LIN {X 0,Y 574.116,Z 389.505,A -85,B 0,C 180,E1 -2265.533,E2 -2265.533} C_VEL
LIN {X 0,Y 574.363,Z 374.82,A -85,B 0,C 180,E1 -2266.255,E2 -2266.255} C_VEL
LIN {X 0,Y 574.533,Z 360.604,A -85,B 0,C 180,E1 -2266.798,E2 -2266.798} C_VEL
LIN {X 0,Y 574.701,Z 345.577,A -85,B 0,C 180,E1 -2267.222,E2 -2267.222} C_VEL
LIN {X 0,Y 574.754,Z 330.659,A -85,B 0,C 180,E1 -2267.503,E2 -2267.503} C_VEL
LIN {X 0,Y 575.181,Z 176.218,A -85,B 0,C 180,E1 -2269.486,E2 -2269.486} C_VEL
LIN {X 0,Y 574.006,Z 169.785,A -85,B 0,C 180,E1 -2269.626,E2 -2269.626} C_VEL
LIN {X 0,Y 574.322,Z 144.284,A -85,B 0,C 180,E1 -2272.673,E2 -2272.673} C_VEL
LIN {X 0,Y 574.579,Z 122.188,A -85,B 0,C 180,E1 -2275.348,E2 -2275.348} C_VEL
LIN {X 0,Y 574.263,Z 119.027,A -85,B 0,C 180,E1 -2275.751,E2 -2275.751} C_VEL
LIN {X 0,Y 573.253,Z 114.708,A -85,B 0,C 180,E1 -2276.341,E2 -2276.341} C_VEL
LIN {X 0,Y 573.234,Z 114.705,A -85,B 0,C 180,E1 -2278.565,E2 -2278.565} C_VEL
LIN {X 0,Y 573.226,Z 114.702,A -85,B 0,C 180,E1 -2280.994,E2 -2280.994} C_VEL
LIN {X 0,Y 573.265,Z 114.701,A -85,B 0,C 180,E1 -2283.524,E2 -2283.524} C_VEL
LIN {X 0,Y 573.216,Z 114.711,A -85,B 0,C 180,E1 -2286.052,E2 -2286.052} C_VEL
LIN {X 0,Y 573.247,Z 114.699,A -85,B 0,C 180,E1 -2288.702,E2 -2288.702} C_VEL
LIN {X 0,Y 573.227,Z 114.709,A -85,B 0,C 180,E1 -2291.593,E2 -2291.593} C_VEL
LIN {X 0,Y 573.227,Z 114.703,A -85,B 0,C 180,E1 -2294.335,E2 -2294.335} C_VEL
LIN {X 0,Y 573.24,Z 114.707,A -85,B 0,C 180,E1 -2297.359,E2 -2297.359} C_VEL
LIN {X 0,Y 573.238,Z 114.699,A -85,B 0,C 180,E1 -2300.392,E2 -2300.392} C_VEL
LIN {X 0,Y 573.255,Z 114.703,A -85,B 0,C 180,E1 -2303.078,E2 -2303.078} C_VEL
LIN {X 0,Y 573.259,Z 114.701,A -85,B 0,C 180,E1 -2305.671,E2 -2305.671} C_VEL
LIN {X 0,Y 573.239,Z 114.699,A -85,B 0,C 180,E1 -2308.185,E2 -2308.185} C_VEL
LIN {X 0,Y 573.245,Z 114.701,A -85,B 0,C 180,E1 -2310.633,E2 -2310.633} C_VEL
LIN {X 0,Y 573.235,Z 114.701,A -85,B 0,C 180,E1 -2313.509,E2 -2313.509} C_VEL
LIN {X 0,Y 573.202,Z 114.704,A -85,B 0,C 180,E1 -2316.133,E2 -2316.133} C_VEL
LIN {X 0,Y 573.248,Z 114.703,A -85,B 0,C 180,E1 -2319.174,E2 -2319.174} C_VEL
LIN {X 0,Y 573.203,Z 114.705,A -85,B 0,C 180,E1 -2321.411,E2 -2321.411} C_VEL
LIN {X 0,Y 573.228,Z 114.7,A -85,B 0,C 180,E1 -2323.621,E2 -2323.621} C_VEL
LIN {X 0,Y 573.244,Z 114.699,A -85,B 0,C 180,E1 -2325.807,E2 -2325.807} C_VEL
LIN {X 0,Y 573.269,Z 114.702,A -85,B 0,C 180,E1 -2328.746,E2 -2328.746} C_VEL
LIN {X 0,Y 573.246,Z 114.698,A -85,B 0,C 180,E1 -2331.54,E2 -2331.54} C_VEL
LIN {X 0,Y 573.276,Z 114.705,A -85,B 0,C 180,E1 -2334.372,E2 -2334.372} C_VEL
LIN {X 0,Y 573.31,Z 114.693,A -85,B 0,C 180,E1 -2337.893,E2 -2337.893} C_VEL
LIN {X 0,Y 573.32,Z 114.692,A -85,B 0,C 180,E1 -2340,E2 -2340} C_VEL
LIN {X 0,Y 573.275,Z 114.695,A -85,B 0,C 180,E1 -2342.811,E2 -2342.811} C_VEL
LIN {X 0,Y 573.268,Z 114.699,A -85,B 0,C 180,E1 -2345.629,E2 -2345.629} C_VEL
LIN {X 0,Y 573.236,Z 114.698,A -85,B 0,C 180,E1 -2348.461,E2 -2348.461} C_VEL
LIN {X 0,Y 573.241,Z 114.699,A -85,B 0,C 180,E1 -2351.313,E2 -2351.313} C_VEL
LIN {X 0,Y 573.241,Z 114.7,A -85,B 0,C 180,E1 -2354.406,E2 -2354.406} C_VEL
LIN {X 0,Y 573.178,Z 114.708,A -85,B 0,C 180,E1 -2357.114,E2 -2357.114} C_VEL
LIN {X 0,Y 573.189,Z 114.708,A -85,B 0,C 180,E1 -2360.079,E2 -2360.079} C_VEL
LIN {X 0,Y 573.188,Z 114.705,A -85,B 0,C 180,E1 -2362.34,E2 -2362.34} C_VEL
LIN {X 0,Y 573.188,Z 114.706,A -85,B 0,C 180,E1 -2364.343,E2 -2364.343} C_VEL
LIN {X 0,Y 572.549,Z 114.789,A -85,B 0,C 180,E1 -2364.929,E2 -2364.929} C_VEL
LIN {X 0,Y 569.719,Z 115.148,A -85,B 0,C 180,E1 -2365.881,E2 -2365.881} C_VEL
LIN {X 0,Y 567.303,Z 115.452,A -85,B 0,C 180,E1 -2366.646,E2 -2366.646} C_VEL
LIN {X 0,Y 566.247,Z 115.579,A -85,B 0,C 180,E1 -2367.237,E2 -2367.237} C_VEL
LIN {X 0,Y 566.152,Z 115.587,A -85,B 0,C 180,E1 -2367.438,E2 -2367.438} C_VEL
LIN {X 0,Y 566.149,Z 115.582,A -85,B 0,C 180,E1 -2369.772,E2 -2369.772} C_VEL
LIN {X 0,Y 566.174,Z 115.579,A -85,B 0,C 180,E1 -2372.424,E2 -2372.424} C_VEL
LIN {X 0,Y 566.159,Z 115.589,A -85,B 0,C 180,E1 -2374.985,E2 -2374.985} C_VEL
LIN {X 0,Y 566.183,Z 115.578,A -85,B 0,C 180,E1 -2377.462,E2 -2377.462} C_VEL
LIN {X 0,Y 566.209,Z 115.574,A -85,B 0,C 180,E1 -2380.199,E2 -2380.199} C_VEL
LIN {X 0,Y 566.154,Z 115.588,A -85,B 0,C 180,E1 -2383.059,E2 -2383.059} C_VEL
LIN {X 0,Y 566.161,Z 115.579,A -85,B 0,C 180,E1 -2386.053,E2 -2386.053} C_VEL
LIN {X 0,Y 566.155,Z 115.589,A -85,B 0,C 180,E1 -2388.858,E2 -2388.858} C_VEL
LIN {X 0,Y 566.203,Z 115.575,A -85,B 0,C 180,E1 -2391.444,E2 -2391.444} C_VEL
LIN {X 0,Y 566.146,Z 115.589,A -85,B 0,C 180,E1 -2394.306,E2 -2394.306} C_VEL
LIN {X 0,Y 566.2,Z 115.577,A -85,B 0,C 180,E1 -2396.896,E2 -2396.896} C_VEL
LIN {X 0,Y 566.173,Z 115.58,A -85,B 0,C 180,E1 -2399.406,E2 -2399.406} C_VEL
LIN {X 0,Y 566.157,Z 115.585,A -85,B 0,C 180,E1 -2401.854,E2 -2401.854} C_VEL
LIN {X 0,Y 566.196,Z 115.586,A -85,B 0,C 180,E1 -2404.25,E2 -2404.25} C_VEL
LIN {X 0,Y 566.168,Z 115.582,A -85,B 0,C 180,E1 -2407.368,E2 -2407.368} C_VEL
LIN {X 0,Y 566.206,Z 115.58,A -85,B 0,C 180,E1 -2409.662,E2 -2409.662} C_VEL
LIN {X 0,Y 566.18,Z 115.585,A -85,B 0,C 180,E1 -2411.921,E2 -2411.921} C_VEL
LIN {X 0,Y 566.193,Z 115.578,A -85,B 0,C 180,E1 -2414.89,E2 -2414.89} C_VEL
LIN {X 0,Y 566.236,Z 115.581,A -85,B 0,C 180,E1 -2417.819,E2 -2417.819} C_VEL
LIN {X 0,Y 566.176,Z 115.586,A -85,B 0,C 180,E1 -2419.992,E2 -2419.992} C_VEL
LIN {X 0,Y 566.216,Z 115.577,A -85,B 0,C 180,E1 -2422.87,E2 -2422.87} C_VEL
LIN {X 0,Y 566.211,Z 115.616,A -85,B 0,C 180,E1 -2425.528,E2 -2425.528} C_VEL
LIN {X 0,Y 567.254,Z 121.648,A -85,B 0,C 180,E1 -2426.448,E2 -2426.448} C_VEL
LIN {X 0,Y 566.93,Z 140.906,A -85,B 0,C 180,E1 -2429.178,E2 -2429.178} C_VEL
LIN {X 0,Y 568.458,Z 149.206,A -85,B 0,C 180,E1 -2429.358,E2 -2429.358} C_VEL
LIN {X 0,Y 567.998,Z 306.402,A -85,B 0,C 180,E1 -2431.418,E2 -2431.418} C_VEL
LIN {X 0,Y 567.821,Z 322.005,A -85,B 0,C 180,E1 -2431.773,E2 -2431.773} C_VEL
LIN {X 0,Y 567.594,Z 336.9,A -85,B 0,C 180,E1 -2432.262,E2 -2432.262} C_VEL
LIN {X 0,Y 567.373,Z 352.096,A -85,B 0,C 180,E1 -2432.929,E2 -2432.929} C_VEL
LIN {X 0,Y 567.124,Z 365.069,A -85,B 0,C 180,E1 -2433.641,E2 -2433.641} C_VEL
LIN {X 0,Y 566.895,Z 378.339,A -85,B 0,C 180,E1 -2434.533,E2 -2434.533} C_VEL
LIN {X 0,Y 566.64,Z 390.468,A -85,B 0,C 180,E1 -2435.516,E2 -2435.516} C_VEL
LIN {X 0,Y 566.457,Z 401.276,A -85,B 0,C 180,E1 -2436.559,E2 -2436.559} C_VEL
LIN {X 0,Y 566.314,Z 410.997,A -85,B 0,C 180,E1 -2437.666,E2 -2437.666} C_VEL
LIN {X 0,Y 566.184,Z 420.325,A -85,B 0,C 180,E1 -2438.926,E2 -2438.926} C_VEL
LIN {X 0,Y 566.046,Z 428.145,A -85,B 0,C 180,E1 -2440.191,E2 -2440.191} C_VEL
LIN {X 0,Y 565.957,Z 434.669,A -85,B 0,C 180,E1 -2441.46,E2 -2441.46} C_VEL
LIN {X 0,Y 565.907,Z 440.687,A -85,B 0,C 180,E1 -2442.917,E2 -2442.917} C_VEL
LIN {X 0,Y 565.884,Z 445.316,A -85,B 0,C 180,E1 -2444.382,E2 -2444.382} C_VEL
LIN {X 0,Y 565.827,Z 448.637,A -85,B 0,C 180,E1 -2445.858,E2 -2445.858} C_VEL
LIN {X 0,Y 565.833,Z 450.67,A -85,B 0,C 180,E1 -2447.343,E2 -2447.343} C_VEL
LIN {X 0,Y 565.852,Z 451.461,A -85,B 0,C 180,E1 -2448.84,E2 -2448.84} C_VEL
LIN {X 0,Y 565.823,Z 450.989,A -85,B 0,C 180,E1 -2450.352,E2 -2450.352} C_VEL
LIN {X 0,Y 565.835,Z 449.211,A -85,B 0,C 180,E1 -2451.877,E2 -2451.877} C_VEL
LIN {X 0,Y 565.894,Z 446.046,A -85,B 0,C 180,E1 -2453.417,E2 -2453.417} C_VEL
LIN {X 0,Y 565.927,Z 441.37,A -85,B 0,C 180,E1 -2454.975,E2 -2454.975} C_VEL
LIN {X 0,Y 565.969,Z 436.799,A -85,B 0,C 180,E1 -2456.156,E2 -2456.156} C_VEL
LIN {X 0,Y 566.03,Z 430.112,A -85,B 0,C 180,E1 -2457.549,E2 -2457.549} C_VEL
LIN {X 0,Y 566.16,Z 421.756,A -85,B 0,C 180,E1 -2458.955,E2 -2458.955} C_VEL
LIN {X 0,Y 566.299,Z 413.022,A -85,B 0,C 180,E1 -2460.173,E2 -2460.173} C_VEL
LIN {X 0,Y 566.444,Z 402.483,A -85,B 0,C 180,E1 -2461.406,E2 -2461.406} C_VEL
LIN {X 0,Y 566.662,Z 390.517,A -85,B 0,C 180,E1 -2462.569,E2 -2462.569} C_VEL
LIN {X 0,Y 566.897,Z 377.894,A -85,B 0,C 180,E1 -2463.589,E2 -2463.589} C_VEL
LIN {X 0,Y 567.109,Z 365.372,A -85,B 0,C 180,E1 -2464.431,E2 -2464.431} C_VEL
LIN {X 0,Y 567.374,Z 352.119,A -85,B 0,C 180,E1 -2465.161,E2 -2465.161} C_VEL
LIN {X 0,Y 567.602,Z 337.434,A -85,B 0,C 180,E1 -2465.806,E2 -2465.806} C_VEL
LIN {X 0,Y 567.825,Z 322.2,A -85,B 0,C 180,E1 -2466.311,E2 -2466.311} C_VEL
LIN {X 0,Y 567.967,Z 306.458,A -85,B 0,C 180,E1 -2466.672,E2 -2466.672} C_VEL
LIN {X 0,Y 568.468,Z 148.223,A -85,B 0,C 180,E1 -2468.745,E2 -2468.745} C_VEL
LIN {X 0,Y 566.907,Z 140.941,A -85,B 0,C 180,E1 -2468.909,E2 -2468.909} C_VEL
LIN {X 0,Y 567.252,Z 121.495,A -85,B 0,C 180,E1 -2471.67,E2 -2471.67} C_VEL
LIN {X 0,Y 566.185,Z 115.588,A -85,B 0,C 180,E1 -2472.599,E2 -2472.599} C_VEL
LIN {X 0,Y 566.166,Z 115.585,A -85,B 0,C 180,E1 -2475.036,E2 -2475.036} C_VEL
LIN {X 0,Y 566.178,Z 115.584,A -85,B 0,C 180,E1 -2477.909,E2 -2477.909} C_VEL
LIN {X 0,Y 566.212,Z 115.582,A -85,B 0,C 180,E1 -2480.726,E2 -2480.726} C_VEL
LIN {X 0,Y 566.184,Z 115.58,A -85,B 0,C 180,E1 -2483.428,E2 -2483.428} C_VEL
LIN {X 0,Y 566.213,Z 115.585,A -85,B 0,C 180,E1 -2486.266,E2 -2486.266} C_VEL
LIN {X 0,Y 566.186,Z 115.579,A -85,B 0,C 180,E1 -2488.924,E2 -2488.924} C_VEL
LIN {X 0,Y 566.192,Z 115.583,A -85,B 0,C 180,E1 -2491.856,E2 -2491.856} C_VEL
LIN {X 0,Y 566.197,Z 115.582,A -85,B 0,C 180,E1 -2494.25,E2 -2494.25} C_VEL
LIN {X 0,Y 566.167,Z 115.58,A -85,B 0,C 180,E1 -2496.72,E2 -2496.72} C_VEL
LIN {X 0,Y 566.206,Z 115.582,A -85,B 0,C 180,E1 -2499.662,E2 -2499.662} C_VEL
LIN {X 0,Y 566.18,Z 115.587,A -85,B 0,C 180,E1 -2501.921,E2 -2501.921} C_VEL
LIN {X 0,Y 566.191,Z 115.577,A -85,B 0,C 180,E1 -2504.89,E2 -2504.89} C_VEL
LIN {X 0,Y 566.234,Z 115.58,A -85,B 0,C 180,E1 -2507.819,E2 -2507.819} C_VEL
LIN {X 0,Y 566.178,Z 115.583,A -85,B 0,C 180,E1 -2509.992,E2 -2509.992} C_VEL
LIN {X 0,Y 566.242,Z 115.572,A -85,B 0,C 180,E1 -2512.87,E2 -2512.87} C_VEL
LIN {X 0,Y 566.277,Z 115.568,A -85,B 0,C 180,E1 -2515.016,E2 -2515.016} C_VEL
LIN {X 0,Y 566.287,Z 115.568,A -85,B 0,C 180,E1 -2517.866,E2 -2517.866} C_VEL
LIN {X 0,Y 566.293,Z 115.566,A -85,B 0,C 180,E1 -2520.711,E2 -2520.711} C_VEL
LIN {X 0,Y 566.263,Z 115.571,A -85,B 0,C 180,E1 -2522.845,E2 -2522.845} C_VEL
LIN {X 0,Y 566.265,Z 115.571,A -85,B 0,C 180,E1 -2525.698,E2 -2525.698} C_VEL
LIN {X 0,Y 566.205,Z 115.577,A -85,B 0,C 180,E1 -2528.566,E2 -2528.566} C_VEL
LIN {X 0,Y 566.243,Z 115.575,A -85,B 0,C 180,E1 -2531.454,E2 -2531.454} C_VEL
LIN {X 0,Y 566.235,Z 115.575,A -85,B 0,C 180,E1 -2534.506,E2 -2534.506} C_VEL
LIN {X 0,Y 566.196,Z 115.581,A -85,B 0,C 180,E1 -2537.331,E2 -2537.331} C_VEL
LIN {X 0,Y 566.206,Z 115.577,A -85,B 0,C 180,E1 -2540.337,E2 -2540.337} C_VEL
LIN {X 0,Y 566.171,Z 115.583,A -85,B 0,C 180,E1 -2543.281,E2 -2543.281} C_VEL
LIN {X 0,Y 566.209,Z 115.575,A -85,B 0,C 180,E1 -2545.749,E2 -2545.749} C_VEL
LIN {X 0,Y 566.202,Z 115.579,A -85,B 0,C 180,E1 -2548.202,E2 -2548.202} C_VEL
LIN {X 0,Y 566.189,Z 115.58,A -85,B 0,C 180,E1 -2551.076,E2 -2551.076} C_VEL
LIN {X 0,Y 566.196,Z 115.578,A -85,B 0,C 180,E1 -2553.732,E2 -2553.732} C_VEL
LIN {X 0,Y 566.199,Z 115.584,A -85,B 0,C 180,E1 -2556.57,E2 -2556.57} C_VEL
LIN {X 0,Y 566.214,Z 115.574,A -85,B 0,C 180,E1 -2559.686,E2 -2559.686} C_VEL
LIN {X 0,Y 566.202,Z 115.576,A -85,B 0,C 180,E1 -2562.917,E2 -2562.917} C_VEL
LIN {X 0,Y 566.198,Z 115.584,A -85,B 0,C 180,E1 -2566.049,E2 -2566.049} C_VEL
LIN {X 0,Y 566.203,Z 115.576,A -85,B 0,C 180,E1 -2569.215,E2 -2569.215} C_VEL
LIN {X 0,Y 566.188,Z 115.582,A -85,B 0,C 180,E1 -2571.637,E2 -2571.637} C_VEL
LIN {X 0,Y 566.161,Z 115.586,A -85,B 0,C 180,E1 -2574.308,E2 -2574.308} C_VEL
LIN {X 0,Y 566.219,Z 115.574,A -85,B 0,C 180,E1 -2576.898,E2 -2576.898} C_VEL
LIN {X 0,Y 566.18,Z 115.583,A -85,B 0,C 180,E1 -2579.407,E2 -2579.407} C_VEL
LIN {X 0,Y 566.211,Z 115.584,A -85,B 0,C 180,E1 -2581.858,E2 -2581.858} C_VEL
LIN {X 0,Y 566.206,Z 115.624,A -85,B 0,C 180,E1 -2583.459,E2 -2583.459} C_VEL
LIN {X 0,Y 567.659,Z 121.967,A -85,B 0,C 180,E1 -2584.322,E2 -2584.322} C_VEL
LIN {X 0,Y 567.503,Z 140.923,A -85,B 0,C 180,E1 -2586.654,E2 -2586.654} C_VEL
LIN {X 0,Y 567.154,Z 164.6,A -85,B 0,C 180,E1 -2589.509,E2 -2589.509} C_VEL
LIN {X 0,Y 567.115,Z 169.895,A -85,B 0,C 180,E1 -2590.142,E2 -2590.142} C_VEL
LIN {X 0,Y 568.508,Z 178.337,A -85,B 0,C 180,E1 -2590.304,E2 -2590.304} C_VEL
LIN {X 0,Y 567.984,Z 335.946,A -85,B 0,C 180,E1 -2592.364,E2 -2592.364} C_VEL
LIN {X 0,Y 567.834,Z 351.709,A -85,B 0,C 180,E1 -2592.72,E2 -2592.72} C_VEL
LIN {X 0,Y 567.616,Z 367.04,A -85,B 0,C 180,E1 -2593.223,E2 -2593.223} C_VEL
LIN {X 0,Y 567.453,Z 380.783,A -85,B 0,C 180,E1 -2593.82,E2 -2593.82} C_VEL
LIN {X 0,Y 567.154,Z 394.255,A -85,B 0,C 180,E1 -2594.549,E2 -2594.549} C_VEL
LIN {X 0,Y 566.931,Z 406.522,A -85,B 0,C 180,E1 -2595.359,E2 -2595.359} C_VEL
LIN {X 0,Y 566.672,Z 419.296,A -85,B 0,C 180,E1 -2596.371,E2 -2596.371} C_VEL
LIN {X 0,Y 566.491,Z 430.752,A -85,B 0,C 180,E1 -2597.461,E2 -2597.461} C_VEL
LIN {X 0,Y 566.268,Z 441.313,A -85,B 0,C 180,E1 -2598.659,E2 -2598.659} C_VEL
LIN {X 0,Y 566.208,Z 449.857,A -85,B 0,C 180,E1 -2599.812,E2 -2599.812} C_VEL
LIN {X 0,Y 566.057,Z 457.737,A -85,B 0,C 180,E1 -2601.072,E2 -2601.072} C_VEL
LIN {X 0,Y 565.997,Z 465.091,A -85,B 0,C 180,E1 -2602.509,E2 -2602.509} C_VEL
LIN {X 0,Y 565.959,Z 470.923,A -85,B 0,C 180,E1 -2603.941,E2 -2603.941} C_VEL
LIN {X 0,Y 565.866,Z 474.387,A -85,B 0,C 180,E1 -2605.013,E2 -2605.013} C_VEL
LIN {X 0,Y 565.91,Z 477.89,A -85,B 0,C 180,E1 -2606.44,E2 -2606.44} C_VEL
LIN {X 0,Y 565.839,Z 480.191,A -85,B 0,C 180,E1 -2607.865,E2 -2607.865} C_VEL
LIN {X 0,Y 565.837,Z 481.349,A -85,B 0,C 180,E1 -2609.289,E2 -2609.289} C_VEL
LIN {X 0,Y 565.837,Z 481.348,A -85,B 0,C 180,E1 -2610.712,E2 -2610.712} C_VEL
LIN {X 0,Y 565.839,Z 480.188,A -85,B 0,C 180,E1 -2612.136,E2 -2612.136} C_VEL
LIN {X 0,Y 565.91,Z 477.885,A -85,B 0,C 180,E1 -2613.56,E2 -2613.56} C_VEL
LIN {X 0,Y 565.867,Z 474.385,A -85,B 0,C 180,E1 -2614.988,E2 -2614.988} C_VEL
LIN {X 0,Y 565.943,Z 469.607,A -85,B 0,C 180,E1 -2616.417,E2 -2616.417} C_VEL
LIN {X 0,Y 566.014,Z 463.42,A -85,B 0,C 180,E1 -2617.85,E2 -2617.85} C_VEL
LIN {X 0,Y 566.071,Z 455.644,A -85,B 0,C 180,E1 -2619.289,E2 -2619.289} C_VEL
LIN {X 0,Y 566.239,Z 447.365,A -85,B 0,C 180,E1 -2620.549,E2 -2620.549} C_VEL
LIN {X 0,Y 566.368,Z 437.388,A -85,B 0,C 180,E1 -2621.815,E2 -2621.815} C_VEL
LIN {X 0,Y 566.586,Z 427.183,A -85,B 0,C 180,E1 -2622.902,E2 -2622.902} C_VEL
LIN {X 0,Y 566.8,Z 415.015,A -85,B 0,C 180,E1 -2623.992,E2 -2623.992} C_VEL
LIN {X 0,Y 567.038,Z 402.332,A -85,B 0,C 180,E1 -2624.937,E2 -2624.937} C_VEL
LIN {X 0,Y 567.235,Z 389.501,A -85,B 0,C 180,E1 -2625.726,E2 -2625.726} C_VEL
LIN {X 0,Y 567.497,Z 374.816,A -85,B 0,C 180,E1 -2626.457,E2 -2626.457} C_VEL
LIN {X 0,Y 567.721,Z 360.603,A -85,B 0,C 180,E1 -2627.006,E2 -2627.006} C_VEL
LIN {X 0,Y 567.923,Z 346.228,A -85,B 0,C 180,E1 -2627.418,E2 -2627.418} C_VEL
LIN {X 0,Y 567.984,Z 331.773,A -85,B 0,C 180,E1 -2627.701,E2 -2627.701} C_VEL
LIN {X 0,Y 568.459,Z 176.883,A -85,B 0,C 180,E1 -2629.717,E2 -2629.717} C_VEL
LIN {X 0,Y 567.12,Z 169.805,A -85,B 0,C 180,E1 -2629.868,E2 -2629.868} C_VEL
LIN {X 0,Y 567.438,Z 145.69,A -85,B 0,C 180,E1 -2632.771,E2 -2632.771} C_VEL
LIN {X 0,Y 567.746,Z 123.819,A -85,B 0,C 180,E1 -2635.451,E2 -2635.451} C_VEL
LIN {X 0,Y 567,Z 118.863,A -85,B 0,C 180,E1 -2636.106,E2 -2636.106} C_VEL
LIN {X 0,Y 566.215,Z 115.583,A -85,B 0,C 180,E1 -2636.584,E2 -2636.584} C_VEL
LIN {X 0,Y 566.189,Z 115.58,A -85,B 0,C 180,E1 -2638.954,E2 -2638.954} C_VEL
LIN {X 0,Y 566.194,Z 115.58,A -85,B 0,C 180,E1 -2641.422,E2 -2641.422} C_VEL
LIN {X 0,Y 566.211,Z 115.585,A -85,B 0,C 180,E1 -2643.956,E2 -2643.956} C_VEL
LIN {X 0,Y 566.201,Z 115.579,A -85,B 0,C 180,E1 -2646.57,E2 -2646.57} C_VEL
LIN {X 0,Y 566.223,Z 115.582,A -85,B 0,C 180,E1 -2649.687,E2 -2649.687} C_VEL
LIN {X 0,Y 566.2,Z 115.577,A -85,B 0,C 180,E1 -2652.917,E2 -2652.917} C_VEL
LIN {X 0,Y 566.197,Z 115.581,A -85,B 0,C 180,E1 -2656.05,E2 -2656.05} C_VEL
LIN {X 0,Y 566.206,Z 115.582,A -85,B 0,C 180,E1 -2659.215,E2 -2659.215} C_VEL
LIN {X 0,Y 566.183,Z 115.584,A -85,B 0,C 180,E1 -2661.637,E2 -2661.637} C_VEL
LIN {X 0,Y 566.164,Z 115.581,A -85,B 0,C 180,E1 -2664.308,E2 -2664.308} C_VEL
LIN {X 0,Y 566.202,Z 115.581,A -85,B 0,C 180,E1 -2666.897,E2 -2666.897} C_VEL
LIN {X 0,Y 566.172,Z 115.585,A -85,B 0,C 180,E1 -2669.407,E2 -2669.407} C_VEL
LIN {X 0,Y 566.173,Z 115.577,A -85,B 0,C 180,E1 -2671.856,E2 -2671.856} C_VEL
LIN {X 0,Y 566.204,Z 115.575,A -85,B 0,C 180,E1 -2674.251,E2 -2674.251} C_VEL
LIN {X 0,Y 566.166,Z 115.583,A -85,B 0,C 180,E1 -2677.368,E2 -2677.368} C_VEL
LIN {X 0,Y 566.204,Z 115.576,A -85,B 0,C 180,E1 -2679.663,E2 -2679.663} C_VEL
LIN {X 0,Y 566.177,Z 115.579,A -85,B 0,C 180,E1 -2681.921,E2 -2681.921} C_VEL
LIN {X 0,Y 566.184,Z 115.58,A -85,B 0,C 180,E1 -2684.152,E2 -2684.152} C_VEL
LIN {X 0,Y 566.171,Z 115.585,A -85,B 0,C 180,E1 -2686.358,E2 -2686.358} C_VEL
LIN {X 0,Y 566.236,Z 115.573,A -85,B 0,C 180,E1 -2689.271,E2 -2689.271} C_VEL
LIN {X 0,Y 566.209,Z 115.58,A -85,B 0,C 180,E1 -2692.153,E2 -2692.153} C_VEL
LIN {X 0,Y 566.256,Z 115.57,A -85,B 0,C 180,E1 -2695.016,E2 -2695.016} C_VEL
LIN {X 0,Y 566.28,Z 115.568,A -85,B 0,C 180,E1 -2697.867,E2 -2697.867} C_VEL
LIN {X 0,Y 566.289,Z 115.567,A -85,B 0,C 180,E1 -2700,E2 -2700} C_VEL
LIN {X 0,Y 566.243,Z 115.571,A -85,B 0,C 180,E1 -2702.846,E2 -2702.846} C_VEL
LIN {X 0,Y 566.237,Z 115.576,A -85,B 0,C 180,E1 -2705.699,E2 -2705.699} C_VEL
LIN {X 0,Y 566.188,Z 115.575,A -85,B 0,C 180,E1 -2708.567,E2 -2708.567} C_VEL
LIN {X 0,Y 566.197,Z 115.577,A -85,B 0,C 180,E1 -2711.456,E2 -2711.456} C_VEL
LIN {X 0,Y 566.188,Z 115.578,A -85,B 0,C 180,E1 -2714.486,E2 -2714.486} C_VEL
LIN {X 0,Y 566.152,Z 115.586,A -85,B 0,C 180,E1 -2717.334,E2 -2717.334} C_VEL
LIN {X 0,Y 566.14,Z 115.584,A -85,B 0,C 180,E1 -2720.34,E2 -2720.34} C_VEL
LIN {X 0,Y 566.135,Z 115.584,A -85,B 0,C 180,E1 -2722.634,E2 -2722.634} C_VEL
LIN {X 0,Y 566.147,Z 115.587,A -85,B 0,C 180,E1 -2725.013,E2 -2725.013} C_VEL
LIN {X 0,Y 566.152,Z 115.587,A -85,B 0,C 180,E1 -2727.438,E2 -2727.438} C_VEL
LIN {X 0,Y 565.458,Z 115.669,A -85,B 0,C 180,E1 -2728.032,E2 -2728.032} C_VEL
LIN {X 0,Y 562.584,Z 116.028,A -85,B 0,C 180,E1 -2728.995,E2 -2728.995} C_VEL
LIN {X 0,Y 560.184,Z 116.324,A -85,B 0,C 180,E1 -2729.771,E2 -2729.771} C_VEL
LIN {X 0,Y 559.173,Z 116.448,A -85,B 0,C 180,E1 -2730.37,E2 -2730.37} C_VEL
LIN {X 0,Y 559.101,Z 116.458,A -85,B 0,C 180,E1 -2730.573,E2 -2730.573} C_VEL
LIN {X 0,Y 559.137,Z 116.458,A -85,B 0,C 180,E1 -2732.717,E2 -2732.717} C_VEL
LIN {X 0,Y 559.114,Z 116.464,A -85,B 0,C 180,E1 -2735.326,E2 -2735.326} C_VEL
LIN {X 0,Y 559.111,Z 116.455,A -85,B 0,C 180,E1 -2738.02,E2 -2738.02} C_VEL
LIN {X 0,Y 559.159,Z 116.452,A -85,B 0,C 180,E1 -2739.941,E2 -2739.941} C_VEL
LIN {X 0,Y 559.105,Z 116.464,A -85,B 0,C 180,E1 -2743.191,E2 -2743.191} C_VEL
LIN {X 0,Y 559.128,Z 116.453,A -85,B 0,C 180,E1 -2745.764,E2 -2745.764} C_VEL
LIN {X 0,Y 559.105,Z 116.462,A -85,B 0,C 180,E1 -2748.224,E2 -2748.224} C_VEL
LIN {X 0,Y 559.172,Z 116.452,A -85,B 0,C 180,E1 -2751.193,E2 -2751.193} C_VEL
LIN {X 0,Y 559.122,Z 116.458,A -85,B 0,C 180,E1 -2753.787,E2 -2753.787} C_VEL
LIN {X 0,Y 559.15,Z 116.463,A -85,B 0,C 180,E1 -2756.424,E2 -2756.424} C_VEL
LIN {X 0,Y 559.154,Z 116.456,A -85,B 0,C 180,E1 -2758.98,E2 -2758.98} C_VEL
LIN {X 0,Y 559.117,Z 116.46,A -85,B 0,C 180,E1 -2761.63,E2 -2761.63} C_VEL
LIN {X 0,Y 559.162,Z 116.459,A -85,B 0,C 180,E1 -2763.902,E2 -2763.902} C_VEL
LIN {X 0,Y 559.117,Z 116.459,A -85,B 0,C 180,E1 -2767.066,E2 -2767.066} C_VEL
LIN {X 0,Y 559.177,Z 116.453,A -85,B 0,C 180,E1 -2769.395,E2 -2769.395} C_VEL
LIN {X 0,Y 559.129,Z 116.462,A -85,B 0,C 180,E1 -2771.685,E2 -2771.685} C_VEL
LIN {X 0,Y 559.144,Z 116.465,A -85,B 0,C 180,E1 -2773.947,E2 -2773.947} C_VEL
LIN {X 0,Y 559.165,Z 116.457,A -85,B 0,C 180,E1 -2776.184,E2 -2776.184} C_VEL
LIN {X 0,Y 559.197,Z 116.452,A -85,B 0,C 180,E1 -2779.133,E2 -2779.133} C_VEL
LIN {X 0,Y 559.195,Z 116.455,A -85,B 0,C 180,E1 -2782.053,E2 -2782.053} C_VEL
LIN {X 0,Y 559.252,Z 116.449,A -85,B 0,C 180,E1 -2784.953,E2 -2784.953} C_VEL
LIN {X 0,Y 559.215,Z 116.594,A -85,B 0,C 180,E1 -2785.337,E2 -2785.337} C_VEL
LIN {X 0,Y 560.328,Z 122.289,A -85,B 0,C 180,E1 -2786.224,E2 -2786.224} C_VEL
LIN {X 0,Y 560.049,Z 141.154,A -85,B 0,C 180,E1 -2788.936,E2 -2788.936} C_VEL
LIN {X 0,Y 561.748,Z 149.207,A -85,B 0,C 180,E1 -2789.111,E2 -2789.111} C_VEL
LIN {X 0,Y 561.251,Z 305.85,A -85,B 0,C 180,E1 -2791.188,E2 -2791.188} C_VEL
LIN {X 0,Y 561.068,Z 321.67,A -85,B 0,C 180,E1 -2791.547,E2 -2791.547} C_VEL
LIN {X 0,Y 560.799,Z 337.211,A -85,B 0,C 180,E1 -2792.065,E2 -2792.065} C_VEL
LIN {X 0,Y 560.541,Z 351.484,A -85,B 0,C 180,E1 -2792.695,E2 -2792.695} C_VEL
LIN {X 0,Y 560.244,Z 364.549,A -85,B 0,C 180,E1 -2793.416,E2 -2793.416} C_VEL
LIN {X 0,Y 560.029,Z 377.892,A -85,B 0,C 180,E1 -2794.318,E2 -2794.318} C_VEL
LIN {X 0,Y 559.712,Z 390.106,A -85,B 0,C 180,E1 -2795.313,E2 -2795.313} C_VEL
LIN {X 0,Y 559.438,Z 402.159,A -85,B 0,C 180,E1 -2796.492,E2 -2796.492} C_VEL
LIN {X 0,Y 559.267,Z 412.938,A -85,B 0,C 180,E1 -2797.764,E2 -2797.764} C_VEL
LIN {X 0,Y 559.104,Z 421.959,A -85,B 0,C 180,E1 -2799.04,E2 -2799.04} C_VEL
LIN {X 0,Y 558.953,Z 429.492,A -85,B 0,C 180,E1 -2800.321,E2 -2800.321} C_VEL
LIN {X 0,Y 558.868,Z 435.753,A -85,B 0,C 180,E1 -2801.607,E2 -2801.607} C_VEL
LIN {X 0,Y 558.819,Z 441.525,A -85,B 0,C 180,E1 -2803.084,E2 -2803.084} C_VEL
LIN {X 0,Y 558.787,Z 445.923,A -85,B 0,C 180,E1 -2804.569,E2 -2804.569} C_VEL
LIN {X 0,Y 558.741,Z 449.031,A -85,B 0,C 180,E1 -2806.064,E2 -2806.064} C_VEL
LIN {X 0,Y 558.748,Z 450.886,A -85,B 0,C 180,E1 -2807.57,E2 -2807.57} C_VEL
LIN {X 0,Y 558.78,Z 451.497,A -85,B 0,C 180,E1 -2809.087,E2 -2809.087} C_VEL
LIN {X 0,Y 558.738,Z 450.819,A -85,B 0,C 180,E1 -2810.621,E2 -2810.621} C_VEL
LIN {X 0,Y 558.749,Z 448.812,A -85,B 0,C 180,E1 -2812.169,E2 -2812.169} C_VEL
LIN {X 0,Y 558.821,Z 445.404,A -85,B 0,C 180,E1 -2813.731,E2 -2813.731} C_VEL
LIN {X 0,Y 558.857,Z 440.469,A -85,B 0,C 180,E1 -2815.313,E2 -2815.313} C_VEL
LIN {X 0,Y 558.918,Z 434.455,A -85,B 0,C 180,E1 -2816.775,E2 -2816.775} C_VEL
LIN {X 0,Y 559.003,Z 427.997,A -85,B 0,C 180,E1 -2818.039,E2 -2818.039} C_VEL
LIN {X 0,Y 559.124,Z 419.913,A -85,B 0,C 180,E1 -2819.355,E2 -2819.355} C_VEL
LIN {X 0,Y 559.297,Z 410.81,A -85,B 0,C 180,E1 -2820.591,E2 -2820.591} C_VEL
LIN {X 0,Y 559.499,Z 399.803,A -85,B 0,C 180,E1 -2821.841,E2 -2821.841} C_VEL
LIN {X 0,Y 559.749,Z 388.032,A -85,B 0,C 180,E1 -2822.955,E2 -2822.955} C_VEL
LIN {X 0,Y 560.033,Z 376.418,A -85,B 0,C 180,E1 -2823.878,E2 -2823.878} C_VEL
LIN {X 0,Y 560.268,Z 364.22,A -85,B 0,C 180,E1 -2824.693,E2 -2824.693} C_VEL
LIN {X 0,Y 560.579,Z 350.088,A -85,B 0,C 180,E1 -2825.462,E2 -2825.462} C_VEL
LIN {X 0,Y 560.793,Z 335.596,A -85,B 0,C 180,E1 -2826.087,E2 -2826.087} C_VEL
LIN {X 0,Y 561.047,Z 320.66,A -85,B 0,C 180,E1 -2826.57,E2 -2826.57} C_VEL
LIN {X 0,Y 561.214,Z 306.017,A -85,B 0,C 180,E1 -2826.9,E2 -2826.9} C_VEL
LIN {X 0,Y 561.786,Z 149.464,A -85,B 0,C 180,E1 -2828.974,E2 -2828.974} C_VEL
LIN {X 0,Y 560.008,Z 141.228,A -85,B 0,C 180,E1 -2829.152,E2 -2829.152} C_VEL
LIN {X 0,Y 560.394,Z 123.75,A -85,B 0,C 180,E1 -2831.658,E2 -2831.658} C_VEL
LIN {X 0,Y 559.526,Z 118.2,A -85,B 0,C 180,E1 -2832.512,E2 -2832.512} C_VEL
LIN {X 0,Y 559.155,Z 116.463,A -85,B 0,C 180,E1 -2832.792,E2 -2832.792} C_VEL
LIN {X 0,Y 559.149,Z 116.458,A -85,B 0,C 180,E1 -2835.761,E2 -2835.761} C_VEL
LIN {X 0,Y 559.157,Z 116.462,A -85,B 0,C 180,E1 -2838.229,E2 -2838.229} C_VEL
LIN {X 0,Y 559.173,Z 116.455,A -85,B 0,C 180,E1 -2841.192,E2 -2841.192} C_VEL
LIN {X 0,Y 559.123,Z 116.462,A -85,B 0,C 180,E1 -2843.787,E2 -2843.787} C_VEL
LIN {X 0,Y 559.164,Z 116.46,A -85,B 0,C 180,E1 -2846.425,E2 -2846.425} C_VEL
LIN {X 0,Y 559.151,Z 116.455,A -85,B 0,C 180,E1 -2848.98,E2 -2848.98} C_VEL
LIN {X 0,Y 559.146,Z 116.457,A -85,B 0,C 180,E1 -2851.623,E2 -2851.623} C_VEL
LIN {X 0,Y 559.163,Z 116.461,A -85,B 0,C 180,E1 -2853.902,E2 -2853.902} C_VEL
LIN {X 0,Y 559.12,Z 116.457,A -85,B 0,C 180,E1 -2857.066,E2 -2857.066} C_VEL
LIN {X 0,Y 559.176,Z 116.454,A -85,B 0,C 180,E1 -2859.395,E2 -2859.395} C_VEL
LIN {X 0,Y 559.129,Z 116.465,A -85,B 0,C 180,E1 -2861.685,E2 -2861.685} C_VEL
LIN {X 0,Y 559.147,Z 116.462,A -85,B 0,C 180,E1 -2863.947,E2 -2863.947} C_VEL
LIN {X 0,Y 559.162,Z 116.457,A -85,B 0,C 180,E1 -2866.183,E2 -2866.183} C_VEL
LIN {X 0,Y 559.196,Z 116.451,A -85,B 0,C 180,E1 -2869.133,E2 -2869.133} C_VEL
LIN {X 0,Y 559.199,Z 116.452,A -85,B 0,C 180,E1 -2872.053,E2 -2872.053} C_VEL
LIN {X 0,Y 559.251,Z 116.443,A -85,B 0,C 180,E1 -2874.953,E2 -2874.953} C_VEL
LIN {X 0,Y 559.258,Z 116.444,A -85,B 0,C 180,E1 -2877.839,E2 -2877.839} C_VEL
LIN {X 0,Y 559.265,Z 116.442,A -85,B 0,C 180,E1 -2880.72,E2 -2880.72} C_VEL
LIN {X 0,Y 559.231,Z 116.447,A -85,B 0,C 180,E1 -2882.881,E2 -2882.881} C_VEL
LIN {X 0,Y 559.233,Z 116.446,A -85,B 0,C 180,E1 -2885.77,E2 -2885.77} C_VEL
LIN {X 0,Y 559.17,Z 116.454,A -85,B 0,C 180,E1 -2888.674,E2 -2888.674} C_VEL
LIN {X 0,Y 559.206,Z 116.449,A -85,B 0,C 180,E1 -2891.6,E2 -2891.6} C_VEL
LIN {X 0,Y 559.201,Z 116.452,A -85,B 0,C 180,E1 -2894.595,E2 -2894.595} C_VEL
LIN {X 0,Y 559.14,Z 116.458,A -85,B 0,C 180,E1 -2897.557,E2 -2897.557} C_VEL
LIN {X 0,Y 559.165,Z 116.452,A -85,B 0,C 180,E1 -2899.837,E2 -2899.837} C_VEL
LIN {X 0,Y 559.14,Z 116.457,A -85,B 0,C 180,E1 -2902.153,E2 -2902.153} C_VEL
LIN {X 0,Y 559.175,Z 116.453,A -85,B 0,C 180,E1 -2905.298,E2 -2905.298} C_VEL
LIN {X 0,Y 559.156,Z 116.454,A -85,B 0,C 180,E1 -2907.713,E2 -2907.713} C_VEL
LIN {X 0,Y 559.15,Z 116.457,A -85,B 0,C 180,E1 -2910.183,E2 -2910.183} C_VEL
LIN {X 0,Y 559.152,Z 116.462,A -85,B 0,C 180,E1 -2912.715,E2 -2912.715} C_VEL
LIN {X 0,Y 559.126,Z 116.458,A -85,B 0,C 180,E1 -2915.324,E2 -2915.324} C_VEL
LIN {X 0,Y 559.132,Z 116.46,A -85,B 0,C 180,E1 -2918.017,E2 -2918.017} C_VEL
LIN {X 0,Y 559.154,Z 116.458,A -85,B 0,C 180,E1 -2920.812,E2 -2920.812} C_VEL
LIN {X 0,Y 559.141,Z 116.455,A -85,B 0,C 180,E1 -2923.734,E2 -2923.734} C_VEL
LIN {X 0,Y 559.145,Z 116.456,A -85,B 0,C 180,E1 -2926.803,E2 -2926.803} C_VEL
LIN {X 0,Y 559.154,Z 116.454,A -85,B 0,C 180,E1 -2929.188,E2 -2929.188} C_VEL
LIN {X 0,Y 559.134,Z 116.466,A -85,B 0,C 180,E1 -2931.983,E2 -2931.983} C_VEL
LIN {X 0,Y 559.13,Z 116.457,A -85,B 0,C 180,E1 -2934.787,E2 -2934.787} C_VEL
LIN {X 0,Y 559.155,Z 116.456,A -85,B 0,C 180,E1 -2937.365,E2 -2937.365} C_VEL
LIN {X 0,Y 559.148,Z 116.462,A -85,B 0,C 180,E1 -2940.143,E2 -2940.143} C_VEL
LIN {X 0,Y 559.169,Z 116.458,A -85,B 0,C 180,E1 -2943.098,E2 -2943.098} C_VEL
LIN {X 0,Y 559.2,Z 116.605,A -85,B 0,C 180,E1 -2943.249,E2 -2943.249} C_VEL
LIN {X 0,Y 560.87,Z 124.322,A -85,B 0,C 180,E1 -2944.308,E2 -2944.308} C_VEL
LIN {X 0,Y 560.558,Z 147.046,A -85,B 0,C 180,E1 -2947.129,E2 -2947.129} C_VEL
LIN {X 0,Y 560.2,Z 169.727,A -85,B 0,C 180,E1 -2949.888,E2 -2949.888} C_VEL
LIN {X 0,Y 561.814,Z 178.899,A -85,B 0,C 180,E1 -2950.07,E2 -2950.07} C_VEL
LIN {X 0,Y 561.231,Z 336.011,A -85,B 0,C 180,E1 -2952.146,E2 -2952.146} C_VEL
LIN {X 0,Y 561.073,Z 351.234,A -85,B 0,C 180,E1 -2952.492,E2 -2952.492} C_VEL
LIN {X 0,Y 560.826,Z 365.805,A -85,B 0,C 180,E1 -2952.967,E2 -2952.967} C_VEL
LIN {X 0,Y 560.615,Z 380.786,A -85,B 0,C 180,E1 -2953.617,E2 -2953.617} C_VEL
LIN {X 0,Y 560.277,Z 394.258,A -85,B 0,C 180,E1 -2954.354,E2 -2954.354} C_VEL
LIN {X 0,Y 559.997,Z 407.305,A -85,B 0,C 180,E1 -2955.23,E2 -2955.23} C_VEL
LIN {X 0,Y 559.697,Z 420.357,A -85,B 0,C 180,E1 -2956.29,E2 -2956.29} C_VEL
LIN {X 0,Y 559.474,Z 432.511,A -85,B 0,C 180,E1 -2957.485,E2 -2957.485} C_VEL
LIN {X 0,Y 559.197,Z 443.245,A -85,B 0,C 180,E1 -2958.758,E2 -2958.758} C_VEL
LIN {X 0,Y 559.091,Z 452.297,A -85,B 0,C 180,E1 -2960.047,E2 -2960.047} C_VEL
LIN {X 0,Y 559,Z 459.751,A -85,B 0,C 180,E1 -2961.323,E2 -2961.323} C_VEL
LIN {X 0,Y 558.899,Z 466.702,A -85,B 0,C 180,E1 -2962.776,E2 -2962.776} C_VEL
LIN {X 0,Y 558.888,Z 472.163,A -85,B 0,C 180,E1 -2964.227,E2 -2964.227} C_VEL
LIN {X 0,Y 558.808,Z 476.292,A -85,B 0,C 180,E1 -2965.673,E2 -2965.673} C_VEL
LIN {X 0,Y 558.793,Z 479.186,A -85,B 0,C 180,E1 -2967.117,E2 -2967.117} C_VEL
LIN {X 0,Y 558.742,Z 480.91,A -85,B 0,C 180,E1 -2968.559,E2 -2968.559} C_VEL
LIN {X 0,Y 558.737,Z 481.5,A -85,B 0,C 180,E1 -2970,E2 -2970} C_VEL
LIN {X 0,Y 558.742,Z 480.908,A -85,B 0,C 180,E1 -2971.442,E2 -2971.442} C_VEL
LIN {X 0,Y 558.793,Z 479.181,A -85,B 0,C 180,E1 -2972.884,E2 -2972.884} C_VEL
LIN {X 0,Y 558.809,Z 476.288,A -85,B 0,C 180,E1 -2974.328,E2 -2974.328} C_VEL
LIN {X 0,Y 558.888,Z 472.164,A -85,B 0,C 180,E1 -2975.774,E2 -2975.774} C_VEL
LIN {X 0,Y 558.9,Z 466.7,A -85,B 0,C 180,E1 -2977.224,E2 -2977.224} C_VEL
LIN {X 0,Y 559.001,Z 459.743,A -85,B 0,C 180,E1 -2978.678,E2 -2978.678} C_VEL
LIN {X 0,Y 559.092,Z 452.29,A -85,B 0,C 180,E1 -2979.953,E2 -2979.953} C_VEL
LIN {X 0,Y 559.228,Z 443.122,A -85,B 0,C 180,E1 -2981.258,E2 -2981.258} C_VEL
LIN {X 0,Y 559.474,Z 432.505,A -85,B 0,C 180,E1 -2982.515,E2 -2982.515} C_VEL
LIN {X 0,Y 559.701,Z 420.355,A -85,B 0,C 180,E1 -2983.71,E2 -2983.71} C_VEL
LIN {X 0,Y 560.006,Z 407.526,A -85,B 0,C 180,E1 -2984.754,E2 -2984.754} C_VEL
LIN {X 0,Y 560.278,Z 394.245,A -85,B 0,C 180,E1 -2985.646,E2 -2985.646} C_VEL
LIN {X 0,Y 560.615,Z 380.765,A -85,B 0,C 180,E1 -2986.384,E2 -2986.384} C_VEL
LIN {X 0,Y 560.832,Z 365.8,A -85,B 0,C 180,E1 -2987.033,E2 -2987.033} C_VEL
LIN {X 0,Y 561.07,Z 350.735,A -85,B 0,C 180,E1 -2987.522,E2 -2987.522} C_VEL
LIN {X 0,Y 561.218,Z 336.27,A -85,B 0,C 180,E1 -2987.85,E2 -2987.85} C_VEL
LIN {X 0,Y 561.777,Z 177.928,A -85,B 0,C 180,E1 -2989.945,E2 -2989.945} C_VEL
LIN {X 0,Y 560.205,Z 169.703,A -85,B 0,C 180,E1 -2990.115,E2 -2990.115} C_VEL
LIN {X 0,Y 560.637,Z 143.941,A -85,B 0,C 180,E1 -2993.259,E2 -2993.259} C_VEL
LIN {X 0,Y 560.873,Z 124.167,A -85,B 0,C 180,E1 -2995.722,E2 -2995.722} C_VEL
LIN {X 0,Y 559.158,Z 116.461,A -85,B 0,C 180,E1 -2996.791,E2 -2996.791} C_VEL
LIN {X 0,Y 559.149,Z 116.463,A -85,B 0,C 180,E1 -2999.858,E2 -2999.858} C_VEL
LIN {X 0,Y 559.158,Z 116.457,A -85,B 0,C 180,E1 -3002.716,E2 -3002.716} C_VEL
LIN {X 0,Y 559.129,Z 116.461,A -85,B 0,C 180,E1 -3005.325,E2 -3005.325} C_VEL
LIN {X 0,Y 559.135,Z 116.464,A -85,B 0,C 180,E1 -3008.018,E2 -3008.018} C_VEL
LIN {X 0,Y 559.157,Z 116.454,A -85,B 0,C 180,E1 -3010.813,E2 -3010.813} C_VEL
LIN {X 0,Y 559.139,Z 116.465,A -85,B 0,C 180,E1 -3013.735,E2 -3013.735} C_VEL
LIN {X 0,Y 559.145,Z 116.457,A -85,B 0,C 180,E1 -3016.804,E2 -3016.804} C_VEL
LIN {X 0,Y 559.158,Z 116.46,A -85,B 0,C 180,E1 -3019.188,E2 -3019.188} C_VEL
LIN {X 0,Y 559.133,Z 116.458,A -85,B 0,C 180,E1 -3021.983,E2 -3021.983} C_VEL
LIN {X 0,Y 559.134,Z 116.459,A -85,B 0,C 180,E1 -3024.788,E2 -3024.788} C_VEL
LIN {X 0,Y 559.155,Z 116.461,A -85,B 0,C 180,E1 -3027.366,E2 -3027.366} C_VEL
LIN {X 0,Y 559.124,Z 116.457,A -85,B 0,C 180,E1 -3030.148,E2 -3030.148} C_VEL
LIN {X 0,Y 559.167,Z 116.458,A -85,B 0,C 180,E1 -3033.175,E2 -3033.175} C_VEL
LIN {X 0,Y 559.119,Z 116.461,A -85,B 0,C 180,E1 -3035.493,E2 -3035.493} C_VEL
LIN {X 0,Y 559.175,Z 116.456,A -85,B 0,C 180,E1 -3038.624,E2 -3038.624} C_VEL
LIN {X 0,Y 559.16,Z 116.461,A -85,B 0,C 180,E1 -3040.926,E2 -3040.926} C_VEL
LIN {X 0,Y 559.144,Z 116.455,A -85,B 0,C 180,E1 -3043.947,E2 -3043.947} C_VEL
LIN {X 0,Y 559.148,Z 116.458,A -85,B 0,C 180,E1 -3046.184,E2 -3046.184} C_VEL
LIN {X 0,Y 559.195,Z 116.451,A -85,B 0,C 180,E1 -3049.134,E2 -3049.134} C_VEL
LIN {X 0,Y 559.183,Z 116.454,A -85,B 0,C 180,E1 -3052.054,E2 -3052.054} C_VEL
LIN {X 0,Y 559.232,Z 116.446,A -85,B 0,C 180,E1 -3054.953,E2 -3054.953} C_VEL
LIN {X 0,Y 559.251,Z 116.443,A -85,B 0,C 180,E1 -3057.84,E2 -3057.84} C_VEL
LIN {X 0,Y 559.258,Z 116.442,A -85,B 0,C 180,E1 -3060,E2 -3060} C_VEL
LIN {X 0,Y 559.211,Z 116.447,A -85,B 0,C 180,E1 -3062.882,E2 -3062.882} C_VEL
LIN {X 0,Y 559.206,Z 116.453,A -85,B 0,C 180,E1 -3065.771,E2 -3065.771} C_VEL
LIN {X 0,Y 559.153,Z 116.45,A -85,B 0,C 180,E1 -3068.675,E2 -3068.675} C_VEL
LIN {X 0,Y 559.158,Z 116.456,A -85,B 0,C 180,E1 -3071.602,E2 -3071.602} C_VEL
LIN {X 0,Y 559.158,Z 116.454,A -85,B 0,C 180,E1 -3074.576,E2 -3074.576} C_VEL
LIN {X 0,Y 559.108,Z 116.467,A -85,B 0,C 180,E1 -3077.559,E2 -3077.559} C_VEL
LIN {X 0,Y 559.1,Z 116.461,A -85,B 0,C 180,E1 -3080.608,E2 -3080.608} C_VEL
LIN {X 0,Y 559.105,Z 116.466,A -85,B 0,C 180,E1 -3083.719,E2 -3083.719} C_VEL
LIN {X 0,Y 559.12,Z 116.458,A -85,B 0,C 180,E1 -3086.101,E2 -3086.101} C_VEL
LIN {X 0,Y 559.102,Z 116.457,A -85,B 0,C 180,E1 -3088.534,E2 -3088.534} C_VEL
LIN {X 0,Y 559.101,Z 116.458,A -85,B 0,C 180,E1 -3090.573,E2 -3090.573} C_VEL
LIN {X 0,Y 558.458,Z 116.545,A -85,B 0,C 180,E1 -3091.174,E2 -3091.174} C_VEL
LIN {X 0,Y 555.606,Z 116.902,A -85,B 0,C 180,E1 -3092.151,E2 -3092.151} C_VEL
LIN {X 0,Y 553.186,Z 117.203,A -85,B 0,C 180,E1 -3092.936,E2 -3092.936} C_VEL
LIN {X 0,Y 552.154,Z 117.33,A -85,B 0,C 180,E1 -3093.543,E2 -3093.543} C_VEL
LIN {X 0,Y 552.075,Z 117.337,A -85,B 0,C 180,E1 -3093.749,E2 -3093.749} C_VEL
LIN {X 0,Y 552.056,Z 117.342,A -85,B 0,C 180,E1 -3096.751,E2 -3096.751} C_VEL
LIN {X 0,Y 552.103,Z 117.332,A -85,B 0,C 180,E1 -3099.53,E2 -3099.53} C_VEL
LIN {X 0,Y 552.088,Z 117.337,A -85,B 0,C 180,E1 -3102.43,E2 -3102.43} C_VEL
LIN {X 0,Y 552.079,Z 117.331,A -85,B 0,C 180,E1 -3105.56,E2 -3105.56} C_VEL
LIN {X 0,Y 552.063,Z 117.344,A -85,B 0,C 180,E1 -3108.548,E2 -3108.548} C_VEL
LIN {X 0,Y 552.115,Z 117.329,A -85,B 0,C 180,E1 -3111.41,E2 -3111.41} C_VEL
LIN {X 0,Y 552.075,Z 117.339,A -85,B 0,C 180,E1 -3114.155,E2 -3114.155} C_VEL
LIN {X 0,Y 552.112,Z 117.33,A -85,B 0,C 180,E1 -3117.155,E2 -3117.155} C_VEL
LIN {X 0,Y 552.1,Z 117.337,A -85,B 0,C 180,E1 -3119.953,E2 -3119.953} C_VEL
LIN {X 0,Y 552.098,Z 117.335,A -85,B 0,C 180,E1 -3123.01,E2 -3123.01} C_VEL
LIN {X 0,Y 552.085,Z 117.343,A -85,B 0,C 180,E1 -3125.961,E2 -3125.961} C_VEL
LIN {X 0,Y 552.121,Z 117.331,A -85,B 0,C 180,E1 -3129.119,E2 -3129.119} C_VEL
LIN {X 0,Y 552.09,Z 117.336,A -85,B 0,C 180,E1 -3131.443,E2 -3131.443} C_VEL
LIN {X 0,Y 552.091,Z 117.339,A -85,B 0,C 180,E1 -3133.736,E2 -3133.736} C_VEL
LIN {X 0,Y 552.133,Z 117.334,A -85,B 0,C 180,E1 -3136.004,E2 -3136.004} C_VEL
LIN {X 0,Y 552.166,Z 117.327,A -85,B 0,C 180,E1 -3138.993,E2 -3138.993} C_VEL
LIN {X 0,Y 552.151,Z 117.334,A -85,B 0,C 180,E1 -3141.951,E2 -3141.951} C_VEL
LIN {X 0,Y 552.191,Z 117.331,A -85,B 0,C 180,E1 -3145.071,E2 -3145.071} C_VEL
LIN {X 0,Y 553.473,Z 124.164,A -85,B 0,C 180,E1 -3146.177,E2 -3146.177} C_VEL
LIN {X 0,Y 553.157,Z 141.353,A -85,B 0,C 180,E1 -3148.676,E2 -3148.676} C_VEL
LIN {X 0,Y 555.12,Z 150.526,A -85,B 0,C 180,E1 -3148.879,E2 -3148.879} C_VEL
LIN {X 0,Y 554.501,Z 306.614,A -85,B 0,C 180,E1 -3150.976,E2 -3150.976} C_VEL
LIN {X 0,Y 554.298,Z 322.215,A -85,B 0,C 180,E1 -3151.339,E2 -3151.339} C_VEL
LIN {X 0,Y 554.014,Z 337.65,A -85,B 0,C 180,E1 -3151.863,E2 -3151.863} C_VEL
LIN {X 0,Y 553.724,Z 350.971,A -85,B 0,C 180,E1 -3152.455,E2 -3152.455} C_VEL
LIN {X 0,Y 553.355,Z 365.614,A -85,B 0,C 180,E1 -3153.276,E2 -3153.276} C_VEL
LIN {X 0,Y 553.103,Z 378.747,A -85,B 0,C 180,E1 -3154.19,E2 -3154.19} C_VEL
LIN {X 0,Y 552.758,Z 390.793,A -85,B 0,C 180,E1 -3155.197,E2 -3155.197} C_VEL
LIN {X 0,Y 552.428,Z 402.711,A -85,B 0,C 180,E1 -3156.391,E2 -3156.391} C_VEL
LIN {X 0,Y 552.246,Z 413.384,A -85,B 0,C 180,E1 -3157.679,E2 -3157.679} C_VEL
LIN {X 0,Y 552.066,Z 422.339,A -85,B 0,C 180,E1 -3158.971,E2 -3158.971} C_VEL
LIN {X 0,Y 551.898,Z 429.821,A -85,B 0,C 180,E1 -3160.269,E2 -3160.269} C_VEL
LIN {X 0,Y 551.805,Z 436.833,A -85,B 0,C 180,E1 -3161.758,E2 -3161.758} C_VEL
LIN {X 0,Y 551.731,Z 442.364,A -85,B 0,C 180,E1 -3163.255,E2 -3163.255} C_VEL
LIN {X 0,Y 551.683,Z 446.53,A -85,B 0,C 180,E1 -3164.761,E2 -3164.761} C_VEL
LIN {X 0,Y 551.642,Z 449.415,A -85,B 0,C 180,E1 -3166.277,E2 -3166.277} C_VEL
LIN {X 0,Y 551.66,Z 451.051,A -85,B 0,C 180,E1 -3167.803,E2 -3167.803} C_VEL
LIN {X 0,Y 551.682,Z 451.41,A -85,B 0,C 180,E1 -3169.488,E2 -3169.488} C_VEL
LIN {X 0,Y 551.641,Z 450.557,A -85,B 0,C 180,E1 -3170.899,E2 -3170.899} C_VEL
LIN {X 0,Y 551.661,Z 448.339,A -85,B 0,C 180,E1 -3172.469,E2 -3172.469} C_VEL
LIN {X 0,Y 551.729,Z 444.692,A -85,B 0,C 180,E1 -3174.055,E2 -3174.055} C_VEL
LIN {X 0,Y 551.754,Z 440.92,A -85,B 0,C 180,E1 -3175.261,E2 -3175.261} C_VEL
LIN {X 0,Y 551.823,Z 435.194,A -85,B 0,C 180,E1 -3176.706,E2 -3176.706} C_VEL
LIN {X 0,Y 551.953,Z 428.261,A -85,B 0,C 180,E1 -3178.107,E2 -3178.107} C_VEL
LIN {X 0,Y 552.097,Z 419.457,A -85,B 0,C 180,E1 -3179.556,E2 -3179.556} C_VEL
LIN {X 0,Y 552.294,Z 410.255,A -85,B 0,C 180,E1 -3180.809,E2 -3180.809} C_VEL
LIN {X 0,Y 552.536,Z 399.291,A -85,B 0,C 180,E1 -3182.059,E2 -3182.059} C_VEL
LIN {X 0,Y 552.81,Z 387.994,A -85,B 0,C 180,E1 -3183.139,E2 -3183.139} C_VEL
LIN {X 0,Y 553.135,Z 375.831,A -85,B 0,C 180,E1 -3184.115,E2 -3184.115} C_VEL
LIN {X 0,Y 553.427,Z 363.147,A -85,B 0,C 180,E1 -3184.963,E2 -3184.963} C_VEL
LIN {X 0,Y 553.782,Z 349.248,A -85,B 0,C 180,E1 -3185.717,E2 -3185.717} C_VEL
LIN {X 0,Y 554.026,Z 335.345,A -85,B 0,C 180,E1 -3186.316,E2 -3186.316} C_VEL
LIN {X 0,Y 554.289,Z 320.966,A -85,B 0,C 180,E1 -3186.786,E2 -3186.786} C_VEL
LIN {X 0,Y 554.484,Z 305.958,A -85,B 0,C 180,E1 -3187.127,E2 -3187.127} C_VEL
LIN {X 0,Y 555.13,Z 150.553,A -85,B 0,C 180,E1 -3189.211,E2 -3189.211} C_VEL
LIN {X 0,Y 553.167,Z 141.365,A -85,B 0,C 180,E1 -3189.423,E2 -3189.423} C_VEL
LIN {X 0,Y 553.508,Z 124.745,A -85,B 0,C 180,E1 -3191.837,E2 -3191.837} C_VEL
LIN {X 0,Y 552.099,Z 117.341,A -85,B 0,C 180,E1 -3193.024,E2 -3193.024} C_VEL
LIN {X 0,Y 552.093,Z 117.336,A -85,B 0,C 180,E1 -3195.562,E2 -3195.562} C_VEL
LIN {X 0,Y 552.11,Z 117.341,A -85,B 0,C 180,E1 -3198.68,E2 -3198.68} C_VEL
LIN {X 0,Y 552.116,Z 117.334,A -85,B 0,C 180,E1 -3201.41,E2 -3201.41} C_VEL
LIN {X 0,Y 552.076,Z 117.345,A -85,B 0,C 180,E1 -3204.155,E2 -3204.155} C_VEL
LIN {X 0,Y 552.117,Z 117.333,A -85,B 0,C 180,E1 -3206.814,E2 -3206.814} C_VEL
LIN {X 0,Y 552.098,Z 117.334,A -85,B 0,C 180,E1 -3209.39,E2 -3209.39} C_VEL
LIN {X 0,Y 552.089,Z 117.339,A -85,B 0,C 180,E1 -3211.9,E2 -3211.9} C_VEL
LIN {X 0,Y 552.088,Z 117.335,A -85,B 0,C 180,E1 -3214.665,E2 -3214.665} C_VEL
LIN {X 0,Y 552.091,Z 117.336,A -85,B 0,C 180,E1 -3217.549,E2 -3217.549} C_VEL
LIN {X 0,Y 552.146,Z 117.33,A -85,B 0,C 180,E1 -3220.375,E2 -3220.375} C_VEL
LIN {X 0,Y 552.119,Z 117.331,A -85,B 0,C 180,E1 -3222.976,E2 -3222.976} C_VEL
LIN {X 0,Y 552.129,Z 117.335,A -85,B 0,C 180,E1 -3226.004,E2 -3226.004} C_VEL
LIN {X 0,Y 552.163,Z 117.326,A -85,B 0,C 180,E1 -3228.993,E2 -3228.993} C_VEL
LIN {X 0,Y 552.155,Z 117.33,A -85,B 0,C 180,E1 -3231.951,E2 -3231.951} C_VEL
LIN {X 0,Y 552.226,Z 117.317,A -85,B 0,C 180,E1 -3234.889,E2 -3234.889} C_VEL
LIN {X 0,Y 552.228,Z 117.32,A -85,B 0,C 180,E1 -3237.812,E2 -3237.812} C_VEL
LIN {X 0,Y 552.236,Z 117.317,A -85,B 0,C 180,E1 -3240.729,E2 -3240.729} C_VEL
LIN {X 0,Y 552.199,Z 117.324,A -85,B 0,C 180,E1 -3242.918,E2 -3242.918} C_VEL
LIN {X 0,Y 552.201,Z 117.322,A -85,B 0,C 180,E1 -3245.844,E2 -3245.844} C_VEL
LIN {X 0,Y 552.141,Z 117.331,A -85,B 0,C 180,E1 -3248.786,E2 -3248.786} C_VEL
LIN {X 0,Y 552.163,Z 117.325,A -85,B 0,C 180,E1 -3251.75,E2 -3251.75} C_VEL
LIN {X 0,Y 552.137,Z 117.334,A -85,B 0,C 180,E1 -3254.748,E2 -3254.748} C_VEL
LIN {X 0,Y 552.097,Z 117.334,A -85,B 0,C 180,E1 -3257.789,E2 -3257.789} C_VEL
LIN {X 0,Y 552.126,Z 117.329,A -85,B 0,C 180,E1 -3260.101,E2 -3260.101} C_VEL
LIN {X 0,Y 552.092,Z 117.338,A -85,B 0,C 180,E1 -3262.451,E2 -3262.451} C_VEL
LIN {X 0,Y 552.155,Z 117.327,A -85,B 0,C 180,E1 -3265.35,E2 -3265.35} C_VEL
LIN {X 0,Y 552.109,Z 117.334,A -85,B 0,C 180,E1 -3268.098,E2 -3268.098} C_VEL
LIN {X 0,Y 552.1,Z 117.342,A -85,B 0,C 180,E1 -3270.609,E2 -3270.609} C_VEL
LIN {X 0,Y 552.106,Z 117.334,A -85,B 0,C 180,E1 -3273.186,E2 -3273.186} C_VEL
LIN {X 0,Y 552.085,Z 117.336,A -85,B 0,C 180,E1 -3275.844,E2 -3275.844} C_VEL
LIN {X 0,Y 552.116,Z 117.335,A -85,B 0,C 180,E1 -3278.589,E2 -3278.589} C_VEL
LIN {X 0,Y 552.12,Z 117.331,A -85,B 0,C 180,E1 -3281.446,E2 -3281.446} C_VEL
LIN {X 0,Y 552.095,Z 117.34,A -85,B 0,C 180,E1 -3284.532,E2 -3284.532} C_VEL
LIN {X 0,Y 552.128,Z 117.33,A -85,B 0,C 180,E1 -3287.585,E2 -3287.585} C_VEL
LIN {X 0,Y 552.133,Z 117.334,A -85,B 0,C 180,E1 -3290.473,E2 -3290.473} C_VEL
LIN {X 0,Y 552.105,Z 117.333,A -85,B 0,C 180,E1 -3293.317,E2 -3293.317} C_VEL
LIN {X 0,Y 552.125,Z 117.338,A -85,B 0,C 180,E1 -3295.939,E2 -3295.939} C_VEL
LIN {X 0,Y 552.118,Z 117.334,A -85,B 0,C 180,E1 -3298.541,E2 -3298.541} C_VEL
LIN {X 0,Y 552.124,Z 117.337,A -85,B 0,C 180,E1 -3301.438,E2 -3301.438} C_VEL
LIN {X 0,Y 552.139,Z 117.341,A -85,B 0,C 180,E1 -3303,E2 -3303} C_VEL
LIN {X 0,Y 554.058,Z 126.238,A -85,B 0,C 180,E1 -3304.238,E2 -3304.238} C_VEL
LIN {X 0,Y 553.684,Z 148.423,A -85,B 0,C 180,E1 -3307.026,E2 -3307.026} C_VEL
LIN {X 0,Y 553.308,Z 169.479,A -85,B 0,C 180,E1 -3309.626,E2 -3309.626} C_VEL
LIN {X 0,Y 555.131,Z 180.201,A -85,B 0,C 180,E1 -3309.84,E2 -3309.84} C_VEL
LIN {X 0,Y 554.468,Z 335.802,A -85,B 0,C 180,E1 -3311.923,E2 -3311.923} C_VEL
LIN {X 0,Y 554.276,Z 351.455,A -85,B 0,C 180,E1 -3312.284,E2 -3312.284} C_VEL
LIN {X 0,Y 553.982,Z 366.847,A -85,B 0,C 180,E1 -3312.798,E2 -3312.798} C_VEL
LIN {X 0,Y 553.78,Z 380.656,A -85,B 0,C 180,E1 -3313.409,E2 -3313.409} C_VEL
LIN {X 0,Y 553.391,Z 394.186,A -85,B 0,C 180,E1 -3314.155,E2 -3314.155} C_VEL
LIN {X 0,Y 553.077,Z 408.149,A -85,B 0,C 180,E1 -3315.103,E2 -3315.103} C_VEL
LIN {X 0,Y 552.76,Z 420.359,A -85,B 0,C 180,E1 -3316.115,E2 -3316.115} C_VEL
LIN {X 0,Y 552.481,Z 432.51,A -85,B 0,C 180,E1 -3317.324,E2 -3317.324} C_VEL
LIN {X 0,Y 552.215,Z 442.485,A -85,B 0,C 180,E1 -3318.514,E2 -3318.514} C_VEL
LIN {X 0,Y 552.124,Z 451.086,A -85,B 0,C 180,E1 -3319.735,E2 -3319.735} C_VEL
LIN {X 0,Y 551.92,Z 458.743,A -85,B 0,C 180,E1 -3321.026,E2 -3321.026} C_VEL
LIN {X 0,Y 551.837,Z 465.09,A -85,B 0,C 180,E1 -3322.315,E2 -3322.315} C_VEL
LIN {X 0,Y 551.769,Z 470.57,A -85,B 0,C 180,E1 -3323.681,E2 -3323.681} C_VEL
LIN {X 0,Y 551.713,Z 474.387,A -85,B 0,C 180,E1 -3324.884,E2 -3324.884} C_VEL
LIN {X 0,Y 551.73,Z 477.888,A -85,B 0,C 180,E1 -3326.349,E2 -3326.349} C_VEL
LIN {X 0,Y 551.655,Z 480.19,A -85,B 0,C 180,E1 -3327.81,E2 -3327.81} C_VEL
LIN {X 0,Y 551.637,Z 481.348,A -85,B 0,C 180,E1 -3329.27,E2 -3329.27} C_VEL
LIN {X 0,Y 551.637,Z 481.347,A -85,B 0,C 180,E1 -3330.73,E2 -3330.73} C_VEL
LIN {X 0,Y 551.655,Z 480.186,A -85,B 0,C 180,E1 -3332.191,E2 -3332.191} C_VEL
LIN {X 0,Y 551.73,Z 477.883,A -85,B 0,C 180,E1 -3333.652,E2 -3333.652} C_VEL
LIN {X 0,Y 551.713,Z 474.386,A -85,B 0,C 180,E1 -3335.116,E2 -3335.116} C_VEL
LIN {X 0,Y 551.82,Z 469.608,A -85,B 0,C 180,E1 -3336.582,E2 -3336.582} C_VEL
LIN {X 0,Y 551.876,Z 463.419,A -85,B 0,C 180,E1 -3338.053,E2 -3338.053} C_VEL
LIN {X 0,Y 551.95,Z 455.641,A -85,B 0,C 180,E1 -3339.528,E2 -3339.528} C_VEL
LIN {X 0,Y 552.184,Z 447.364,A -85,B 0,C 180,E1 -3340.821,E2 -3340.821} C_VEL
LIN {X 0,Y 552.353,Z 437.388,A -85,B 0,C 180,E1 -3342.119,E2 -3342.119} C_VEL
LIN {X 0,Y 552.609,Z 427.18,A -85,B 0,C 180,E1 -3343.234,E2 -3343.234} C_VEL
LIN {X 0,Y 552.908,Z 415.013,A -85,B 0,C 180,E1 -3344.352,E2 -3344.352} C_VEL
LIN {X 0,Y 553.25,Z 402.407,A -85,B 0,C 180,E1 -3345.31,E2 -3345.31} C_VEL
LIN {X 0,Y 553.517,Z 389.411,A -85,B 0,C 180,E1 -3346.126,E2 -3346.126} C_VEL
LIN {X 0,Y 553.846,Z 374.666,A -85,B 0,C 180,E1 -3346.875,E2 -3346.875} C_VEL
LIN {X 0,Y 554.143,Z 360.404,A -85,B 0,C 180,E1 -3347.436,E2 -3347.436} C_VEL
LIN {X 0,Y 554.365,Z 345.912,A -85,B 0,C 180,E1 -3347.86,E2 -3347.86} C_VEL
LIN {X 0,Y 554.478,Z 330.953,A -85,B 0,C 180,E1 -3348.155,E2 -3348.155} C_VEL
LIN {X 0,Y 555.147,Z 179.862,A -85,B 0,C 180,E1 -3350.164,E2 -3350.164} C_VEL
LIN {X 0,Y 553.28,Z 169.42,A -85,B 0,C 180,E1 -3350.389,E2 -3350.389} C_VEL
LIN {X 0,Y 553.751,Z 145.346,A -85,B 0,C 180,E1 -3353.367,E2 -3353.367} C_VEL
LIN {X 0,Y 554.074,Z 126.311,A -85,B 0,C 180,E1 -3355.766,E2 -3355.766} C_VEL
LIN {X 0,Y 552.131,Z 117.336,A -85,B 0,C 180,E1 -3357.033,E2 -3357.033} C_VEL
LIN {X 0,Y 552.118,Z 117.339,A -85,B 0,C 180,E1 -3360.051,E2 -3360.051} C_VEL
LIN {X 0,Y 552.116,Z 117.334,A -85,B 0,C 180,E1 -3362.847,E2 -3362.847} C_VEL
LIN {X 0,Y 552.078,Z 117.341,A -85,B 0,C 180,E1 -3365.44,E2 -3365.44} C_VEL
LIN {X 0,Y 552.099,Z 117.341,A -85,B 0,C 180,E1 -3367.886,E2 -3367.886} C_VEL
LIN {X 0,Y 552.112,Z 117.333,A -85,B 0,C 180,E1 -3370.482,E2 -3370.482} C_VEL
LIN {X 0,Y 552.094,Z 117.341,A -85,B 0,C 180,E1 -3373.482,E2 -3373.482} C_VEL
LIN {X 0,Y 552.109,Z 117.333,A -85,B 0,C 180,E1 -3376.577,E2 -3376.577} C_VEL
LIN {X 0,Y 552.11,Z 117.34,A -85,B 0,C 180,E1 -3379.519,E2 -3379.519} C_VEL
LIN {X 0,Y 552.093,Z 117.334,A -85,B 0,C 180,E1 -3382.336,E2 -3382.336} C_VEL
LIN {X 0,Y 552.085,Z 117.34,A -85,B 0,C 180,E1 -3385.051,E2 -3385.051} C_VEL
LIN {X 0,Y 552.115,Z 117.334,A -85,B 0,C 180,E1 -3387.682,E2 -3387.682} C_VEL
LIN {X 0,Y 552.089,Z 117.334,A -85,B 0,C 180,E1 -3390.234,E2 -3390.234} C_VEL
LIN {X 0,Y 552.133,Z 117.332,A -85,B 0,C 180,E1 -3393.002,E2 -3393.002} C_VEL
LIN {X 0,Y 552.082,Z 117.335,A -85,B 0,C 180,E1 -3395.961,E2 -3395.961} C_VEL
LIN {X 0,Y 552.119,Z 117.336,A -85,B 0,C 180,E1 -3399.12,E2 -3399.12} C_VEL
LIN {X 0,Y 552.087,Z 117.335,A -85,B 0,C 180,E1 -3401.443,E2 -3401.443} C_VEL
LIN {X 0,Y 552.094,Z 117.333,A -85,B 0,C 180,E1 -3403.737,E2 -3403.737} C_VEL
LIN {X 0,Y 552.111,Z 117.333,A -85,B 0,C 180,E1 -3406.004,E2 -3406.004} C_VEL
LIN {X 0,Y 552.164,Z 117.328,A -85,B 0,C 180,E1 -3408.994,E2 -3408.994} C_VEL
LIN {X 0,Y 552.141,Z 117.33,A -85,B 0,C 180,E1 -3411.952,E2 -3411.952} C_VEL
LIN {X 0,Y 552.209,Z 117.321,A -85,B 0,C 180,E1 -3414.889,E2 -3414.889} C_VEL
LIN {X 0,Y 552.222,Z 117.318,A -85,B 0,C 180,E1 -3417.812,E2 -3417.812} C_VEL
LIN {X 0,Y 552.226,Z 117.317,A -85,B 0,C 180,E1 -3420,E2 -3420} C_VEL
LIN {X 0,Y 552.179,Z 117.323,A -85,B 0,C 180,E1 -3422.919,E2 -3422.919} C_VEL
LIN {X 0,Y 552.176,Z 117.33,A -85,B 0,C 180,E1 -3425.844,E2 -3425.844} C_VEL
LIN {X 0,Y 552.126,Z 117.324,A -85,B 0,C 180,E1 -3428.787,E2 -3428.787} C_VEL
LIN {X 0,Y 552.102,Z 117.337,A -85,B 0,C 180,E1 -3431.752,E2 -3431.752} C_VEL
LIN {X 0,Y 552.094,Z 117.333,A -85,B 0,C 180,E1 -3434.75,E2 -3434.75} C_VEL
LIN {X 0,Y 552.069,Z 117.344,A -85,B 0,C 180,E1 -3437.79,E2 -3437.79} C_VEL
LIN {X 0,Y 552.047,Z 117.341,A -85,B 0,C 180,E1 -3440.105,E2 -3440.105} C_VEL
LIN {X 0,Y 552.039,Z 117.339,A -85,B 0,C 180,E1 -3442.454,E2 -3442.454} C_VEL
LIN {X 0,Y 552.067,Z 117.345,A -85,B 0,C 180,E1 -3445.33,E2 -3445.33} C_VEL
LIN {X 0,Y 552.051,Z 117.335,A -85,B 0,C 180,E1 -3448.102,E2 -3448.102} C_VEL
LIN {X 0,Y 552.071,Z 117.333,A -85,B 0,C 180,E1 -3450.612,E2 -3450.612} C_VEL
LIN {X 0,Y 552.092,Z 117.343,A -85,B 0,C 180,E1 -3453.188,E2 -3453.188} C_VEL
LIN {X 0,Y 552.075,Z 117.337,A -85,B 0,C 180,E1 -3453.749,E2 -3453.749} C_VEL
LIN {X 0,Y 551.419,Z 117.418,A -85,B 0,C 180,E1 -3454.358,E2 -3454.358} C_VEL
LIN {X 0,Y 548.557,Z 117.783,A -85,B 0,C 180,E1 -3455.346,E2 -3455.346} C_VEL
LIN {X 0,Y 546.13,Z 118.089,A -85,B 0,C 180,E1 -3456.141,E2 -3456.141} C_VEL
LIN {X 0,Y 545.088,Z 118.215,A -85,B 0,C 180,E1 -3456.755,E2 -3456.755} C_VEL
LIN {X 0,Y 545.004,Z 118.222,A -85,B 0,C 180,E1 -3456.963,E2 -3456.963} C_VEL
LIN {X 0,Y 545.051,Z 118.213,A -85,B 0,C 180,E1 -3459.316,E2 -3459.316} C_VEL
LIN {X 0,Y 545.037,Z 118.213,A -85,B 0,C 180,E1 -3462.107,E2 -3462.107} C_VEL
LIN {X 0,Y 545.026,Z 118.213,A -85,B 0,C 180,E1 -3465.172,E2 -3465.172} C_VEL
LIN {X 0,Y 545.037,Z 118.212,A -85,B 0,C 180,E1 -3467.893,E2 -3467.893} C_VEL
LIN {X 0,Y 545.078,Z 118.212,A -85,B 0,C 180,E1 -3470.818,E2 -3470.818} C_VEL
LIN {X 0,Y 545.037,Z 118.212,A -85,B 0,C 180,E1 -3473.619,E2 -3473.619} C_VEL
LIN {X 0,Y 545.051,Z 118.219,A -85,B 0,C 180,E1 -3476.327,E2 -3476.327} C_VEL
LIN {X 0,Y 545.068,Z 118.211,A -85,B 0,C 180,E1 -3478.952,E2 -3478.952} C_VEL
LIN {X 0,Y 545.046,Z 118.212,A -85,B 0,C 180,E1 -3481.504,E2 -3481.504} C_VEL
LIN {X 0,Y 545.049,Z 118.219,A -85,B 0,C 180,E1 -3483.997,E2 -3483.997} C_VEL
LIN {X 0,Y 545.076,Z 118.213,A -85,B 0,C 180,E1 -3486.44,E2 -3486.44} C_VEL
LIN {X 0,Y 545.096,Z 118.21,A -85,B 0,C 180,E1 -3489.628,E2 -3489.628} C_VEL
LIN {X 0,Y 545.059,Z 118.209,A -85,B 0,C 180,E1 -3492.748,E2 -3492.748} C_VEL
LIN {X 0,Y 545.088,Z 118.212,A -85,B 0,C 180,E1 -3495.819,E2 -3495.819} C_VEL
LIN {X 0,Y 545.123,Z 118.204,A -85,B 0,C 180,E1 -3498.849,E2 -3498.849} C_VEL
LIN {X 0,Y 545.099,Z 118.213,A -85,B 0,C 180,E1 -3501.846,E2 -3501.846} C_VEL
LIN {X 0,Y 545.197,Z 118.29,A -85,B 0,C 180,E1 -3504.892,E2 -3504.892} C_VEL
LIN {X 0,Y 546.613,Z 126.041,A -85,B 0,C 180,E1 -3506.129,E2 -3506.129} C_VEL
LIN {X 0,Y 546.285,Z 141.56,A -85,B 0,C 180,E1 -3508.41,E2 -3508.41} C_VEL
LIN {X 0,Y 548.47,Z 152.238,A -85,B 0,C 180,E1 -3508.644,E2 -3508.644} C_VEL
LIN {X 0,Y 547.762,Z 306.127,A -85,B 0,C 180,E1 -3510.735,E2 -3510.735} C_VEL
LIN {X 0,Y 547.555,Z 321.981,A -85,B 0,C 180,E1 -3511.103,E2 -3511.103} C_VEL
LIN {X 0,Y 547.26,Z 336.976,A -85,B 0,C 180,E1 -3511.609,E2 -3511.609} C_VEL
LIN {X 0,Y 546.922,Z 350.436,A -85,B 0,C 180,E1 -3512.209,E2 -3512.209} C_VEL
LIN {X 0,Y 546.548,Z 365.244,A -85,B 0,C 180,E1 -3513.04,E2 -3513.04} C_VEL
LIN {X 0,Y 546.212,Z 378.502,A -85,B 0,C 180,E1 -3513.965,E2 -3513.965} C_VEL
LIN {X 0,Y 545.842,Z 390.607,A -85,B 0,C 180,E1 -3514.986,E2 -3514.986} C_VEL
LIN {X 0,Y 545.574,Z 401.665,A -85,B 0,C 180,E1 -3516.1,E2 -3516.1} C_VEL
LIN {X 0,Y 545.28,Z 411.253,A -85,B 0,C 180,E1 -3517.243,E2 -3517.243} C_VEL
LIN {X 0,Y 545.027,Z 420.345,A -85,B 0,C 180,E1 -3518.528,E2 -3518.528} C_VEL
LIN {X 0,Y 544.875,Z 428.122,A -85,B 0,C 180,E1 -3519.84,E2 -3519.84} C_VEL
LIN {X 0,Y 544.726,Z 435.342,A -85,B 0,C 180,E1 -3521.318,E2 -3521.318} C_VEL
LIN {X 0,Y 544.668,Z 440.666,A -85,B 0,C 180,E1 -3522.671,E2 -3522.671} C_VEL
LIN {X 0,Y 544.627,Z 445.296,A -85,B 0,C 180,E1 -3524.192,E2 -3524.192} C_VEL
LIN {X 0,Y 544.547,Z 448.622,A -85,B 0,C 180,E1 -3525.725,E2 -3525.725} C_VEL
LIN {X 0,Y 544.578,Z 450.662,A -85,B 0,C 180,E1 -3527.267,E2 -3527.267} C_VEL
LIN {X 0,Y 544.554,Z 451.459,A -85,B 0,C 180,E1 -3528.823,E2 -3528.823} C_VEL
LIN {X 0,Y 544.527,Z 450.993,A -85,B 0,C 180,E1 -3530.394,E2 -3530.394} C_VEL
LIN {X 0,Y 544.547,Z 449.221,A -85,B 0,C 180,E1 -3531.979,E2 -3531.979} C_VEL
LIN {X 0,Y 544.625,Z 445.963,A -85,B 0,C 180,E1 -3533.621,E2 -3533.621} C_VEL
LIN {X 0,Y 544.665,Z 441.388,A -85,B 0,C 180,E1 -3535.202,E2 -3535.202} C_VEL
LIN {X 0,Y 544.733,Z 436.819,A -85,B 0,C 180,E1 -3536.43,E2 -3536.43} C_VEL
LIN {X 0,Y 544.828,Z 430.131,A -85,B 0,C 180,E1 -3537.879,E2 -3537.879} C_VEL
LIN {X 0,Y 545.005,Z 421.79,A -85,B 0,C 180,E1 -3539.342,E2 -3539.342} C_VEL
LIN {X 0,Y 545.227,Z 413.084,A -85,B 0,C 180,E1 -3540.612,E2 -3540.612} C_VEL
LIN {X 0,Y 545.491,Z 402.645,A -85,B 0,C 180,E1 -3541.886,E2 -3541.886} C_VEL
LIN {X 0,Y 545.805,Z 391.318,A -85,B 0,C 180,E1 -3543.04,E2 -3543.04} C_VEL
LIN {X 0,Y 546.14,Z 379.586,A -85,B 0,C 180,E1 -3544.04,E2 -3544.04} C_VEL
LIN {X 0,Y 546.46,Z 367.197,A -85,B 0,C 180,E1 -3544.924,E2 -3544.924} C_VEL
LIN {X 0,Y 546.847,Z 353.634,A -85,B 0,C 180,E1 -3545.717,E2 -3545.717} C_VEL
LIN {X 0,Y 547.179,Z 339.265,A -85,B 0,C 180,E1 -3546.387,E2 -3546.387} C_VEL
LIN {X 0,Y 547.488,Z 324.6,A -85,B 0,C 180,E1 -3546.907,E2 -3546.907} C_VEL
LIN {X 0,Y 547.701,Z 309.413,A -85,B 0,C 180,E1 -3547.29,E2 -3547.29} C_VEL
LIN {X 0,Y 547.828,Z 288.457,A -85,B 0,C 180,E1 -3547.611,E2 -3547.611} C_VEL
LIN {X 0,Y 548.423,Z 151.23,A -85,B 0,C 180,E1 -3549.462,E2 -3549.462} C_VEL
LIN {X 0,Y 546.29,Z 141.551,A -85,B 0,C 180,E1 -3549.696,E2 -3549.696} C_VEL
LIN {X 0,Y 546.658,Z 126.206,A -85,B 0,C 180,E1 -3551.953,E2 -3551.953} C_VEL
LIN {X 0,Y 545.039,Z 118.219,A -85,B 0,C 180,E1 -3553.264,E2 -3553.264} C_VEL
LIN {X 0,Y 545.051,Z 118.219,A -85,B 0,C 180,E1 -3556.226,E2 -3556.226} C_VEL
LIN {X 0,Y 545.074,Z 118.215,A -85,B 0,C 180,E1 -3558.884,E2 -3558.884} C_VEL
LIN {X 0,Y 545.079,Z 118.214,A -85,B 0,C 180,E1 -3560.818,E2 -3560.818} C_VEL
LIN {X 0,Y 545.036,Z 118.216,A -85,B 0,C 180,E1 -3563.619,E2 -3563.619} C_VEL
LIN {X 0,Y 545.067,Z 118.218,A -85,B 0,C 180,E1 -3566.328,E2 -3566.328} C_VEL
LIN {X 0,Y 545.065,Z 118.21,A -85,B 0,C 180,E1 -3568.952,E2 -3568.952} C_VEL
LIN {X 0,Y 545.082,Z 118.208,A -85,B 0,C 180,E1 -3571.506,E2 -3571.506} C_VEL
LIN {X 0,Y 545.063,Z 118.219,A -85,B 0,C 180,E1 -3573.998,E2 -3573.998} C_VEL
LIN {X 0,Y 545.035,Z 118.212,A -85,B 0,C 180,E1 -3577.242,E2 -3577.242} C_VEL
LIN {X 0,Y 545.118,Z 118.205,A -85,B 0,C 180,E1 -3580.414,E2 -3580.414} C_VEL
LIN {X 0,Y 545.048,Z 118.216,A -85,B 0,C 180,E1 -3583.52,E2 -3583.52} C_VEL
LIN {X 0,Y 545.084,Z 118.216,A -85,B 0,C 180,E1 -3585.819,E2 -3585.819} C_VEL
LIN {X 0,Y 545.119,Z 118.203,A -85,B 0,C 180,E1 -3588.849,E2 -3588.849} C_VEL
LIN {X 0,Y 545.126,Z 118.208,A -85,B 0,C 180,E1 -3591.847,E2 -3591.847} C_VEL
LIN {X 0,Y 545.202,Z 118.191,A -85,B 0,C 180,E1 -3594.823,E2 -3594.823} C_VEL
LIN {X 0,Y 545.2,Z 118.196,A -85,B 0,C 180,E1 -3597.783,E2 -3597.783} C_VEL
LIN {X 0,Y 545.208,Z 118.193,A -85,B 0,C 180,E1 -3600.738,E2 -3600.738} C_VEL
LIN {X 0,Y 545.166,Z 118.2,A -85,B 0,C 180,E1 -3602.956,E2 -3602.956} C_VEL
LIN {X 0,Y 545.171,Z 118.197,A -85,B 0,C 180,E1 -3605.919,E2 -3605.919} C_VEL
LIN {X 0,Y 545.102,Z 118.21,A -85,B 0,C 180,E1 -3608.9,E2 -3608.9} C_VEL
LIN {X 0,Y 545.135,Z 118.2,A -85,B 0,C 180,E1 -3611.904,E2 -3611.904} C_VEL
LIN {X 0,Y 545.085,Z 118.216,A -85,B 0,C 180,E1 -3614.943,E2 -3614.943} C_VEL
LIN {X 0,Y 545.069,Z 118.209,A -85,B 0,C 180,E1 -3618.026,E2 -3618.026} C_VEL
LIN {X 0,Y 545.092,Z 118.207,A -85,B 0,C 180,E1 -3620.372,E2 -3620.372} C_VEL
LIN {X 0,Y 545.08,Z 118.208,A -85,B 0,C 180,E1 -3623.559,E2 -3623.559} C_VEL
LIN {X 0,Y 545.078,Z 118.208,A -85,B 0,C 180,E1 -3626,E2 -3626} C_VEL
LIN {X 0,Y 545.088,Z 118.213,A -85,B 0,C 180,E1 -3628.748,E2 -3628.748} C_VEL
LIN {X 0,Y 545.057,Z 118.21,A -85,B 0,C 180,E1 -3631.679,E2 -3631.679} C_VEL
LIN {X 0,Y 545.058,Z 118.218,A -85,B 0,C 180,E1 -3634.565,E2 -3634.565} C_VEL
LIN {X 0,Y 545.035,Z 118.213,A -85,B 0,C 180,E1 -3637.304,E2 -3637.304} C_VEL
LIN {X 0,Y 545.064,Z 118.213,A -85,B 0,C 180,E1 -3640.143,E2 -3640.143} C_VEL
LIN {X 0,Y 545.077,Z 118.205,A -85,B 0,C 180,E1 -3643.107,E2 -3643.107} C_VEL
LIN {X 0,Y 545.066,Z 118.215,A -85,B 0,C 180,E1 -3646.224,E2 -3646.224} C_VEL
LIN {X 0,Y 545.08,Z 118.209,A -85,B 0,C 180,E1 -3648.885,E2 -3648.885} C_VEL
LIN {X 0,Y 545.083,Z 118.21,A -85,B 0,C 180,E1 -3650.819,E2 -3650.819} C_VEL
LIN {X 0,Y 545.041,Z 118.216,A -85,B 0,C 180,E1 -3653.62,E2 -3653.62} C_VEL
LIN {X 0,Y 545.065,Z 118.214,A -85,B 0,C 180,E1 -3656.328,E2 -3656.328} C_VEL
LIN {X 0,Y 545.065,Z 118.211,A -85,B 0,C 180,E1 -3658.952,E2 -3658.952} C_VEL
LIN {X 0,Y 545.102,Z 118.213,A -85,B 0,C 180,E1 -3661.508,E2 -3661.508} C_VEL
LIN {X 0,Y 545.109,Z 118.219,A -85,B 0,C 180,E1 -3662.762,E2 -3662.762} C_VEL
LIN {X 0,Y 547.194,Z 127.714,A -85,B 0,C 180,E1 -3664.108,E2 -3664.108} C_VEL
LIN {X 0,Y 546.812,Z 148.204,A -85,B 0,C 180,E1 -3666.721,E2 -3666.721} C_VEL
LIN {X 0,Y 546.391,Z 169.244,A -85,B 0,C 180,E1 -3669.354,E2 -3669.354} C_VEL
LIN {X 0,Y 548.47,Z 180.925,A -85,B 0,C 180,E1 -3669.597,E2 -3669.597} C_VEL
LIN {X 0,Y 547.701,Z 335.446,A -85,B 0,C 180,E1 -3671.691,E2 -3671.691} C_VEL
LIN {X 0,Y 547.503,Z 351.178,A -85,B 0,C 180,E1 -3672.057,E2 -3672.057} C_VEL
LIN {X 0,Y 547.184,Z 366.59,A -85,B 0,C 180,E1 -3672.577,E2 -3672.577} C_VEL
LIN {X 0,Y 546.918,Z 380.405,A -85,B 0,C 180,E1 -3673.194,E2 -3673.194} C_VEL
LIN {X 0,Y 546.504,Z 393.943,A -85,B 0,C 180,E1 -3673.95,E2 -3673.95} C_VEL
LIN {X 0,Y 546.129,Z 407.917,A -85,B 0,C 180,E1 -3674.909,E2 -3674.909} C_VEL
LIN {X 0,Y 545.786,Z 420.199,A -85,B 0,C 180,E1 -3675.934,E2 -3675.934} C_VEL
LIN {X 0,Y 545.491,Z 432.432,A -85,B 0,C 180,E1 -3677.159,E2 -3677.159} C_VEL
LIN {X 0,Y 545.174,Z 443.1,A -85,B 0,C 180,E1 -3678.446,E2 -3678.446} C_VEL
LIN {X 0,Y 545.05,Z 452.298,A -85,B 0,C 180,E1 -3679.788,E2 -3679.788} C_VEL
LIN {X 0,Y 544.845,Z 459.75,A -85,B 0,C 180,E1 -3681.096,E2 -3681.096} C_VEL
LIN {X 0,Y 544.744,Z 466.701,A -85,B 0,C 180,E1 -3682.588,E2 -3682.588} C_VEL
LIN {X 0,Y 544.709,Z 472.163,A -85,B 0,C 180,E1 -3684.076,E2 -3684.076} C_VEL
LIN {X 0,Y 544.606,Z 476.291,A -85,B 0,C 180,E1 -3685.56,E2 -3685.56} C_VEL
LIN {X 0,Y 544.643,Z 479.184,A -85,B 0,C 180,E1 -3687.042,E2 -3687.042} C_VEL
LIN {X 0,Y 544.543,Z 480.909,A -85,B 0,C 180,E1 -3688.521,E2 -3688.521} C_VEL
LIN {X 0,Y 544.538,Z 481.5,A -85,B 0,C 180,E1 -3690,E2 -3690} C_VEL
LIN {X 0,Y 544.543,Z 480.907,A -85,B 0,C 180,E1 -3691.479,E2 -3691.479} C_VEL
LIN {X 0,Y 544.643,Z 479.179,A -85,B 0,C 180,E1 -3692.959,E2 -3692.959} C_VEL
LIN {X 0,Y 544.606,Z 476.287,A -85,B 0,C 180,E1 -3694.441,E2 -3694.441} C_VEL
LIN {X 0,Y 544.709,Z 472.164,A -85,B 0,C 180,E1 -3695.925,E2 -3695.925} C_VEL
LIN {X 0,Y 544.745,Z 466.699,A -85,B 0,C 180,E1 -3697.413,E2 -3697.413} C_VEL
LIN {X 0,Y 544.845,Z 459.741,A -85,B 0,C 180,E1 -3698.905,E2 -3698.905} C_VEL
LIN {X 0,Y 545.074,Z 451.078,A -85,B 0,C 180,E1 -3700.4,E2 -3700.4} C_VEL
LIN {X 0,Y 545.237,Z 441.689,A -85,B 0,C 180,E1 -3701.735,E2 -3701.735} C_VEL
LIN {X 0,Y 545.492,Z 432.43,A -85,B 0,C 180,E1 -3702.841,E2 -3702.841} C_VEL
LIN {X 0,Y 545.797,Z 420.208,A -85,B 0,C 180,E1 -3704.067,E2 -3704.067} C_VEL
LIN {X 0,Y 546.15,Z 407.705,A -85,B 0,C 180,E1 -3705.108,E2 -3705.108} C_VEL
LIN {X 0,Y 546.506,Z 393.952,A -85,B 0,C 180,E1 -3706.051,E2 -3706.051} C_VEL
LIN {X 0,Y 546.896,Z 380.411,A -85,B 0,C 180,E1 -3706.807,E2 -3706.807} C_VEL
LIN {X 0,Y 547.191,Z 366.62,A -85,B 0,C 180,E1 -3707.423,E2 -3707.423} C_VEL
LIN {X 0,Y 547.501,Z 351.217,A -85,B 0,C 180,E1 -3707.944,E2 -3707.944} C_VEL
LIN {X 0,Y 547.696,Z 335.556,A -85,B 0,C 180,E1 -3708.308,E2 -3708.308} C_VEL
LIN {X 0,Y 548.459,Z 180.937,A -85,B 0,C 180,E1 -3710.404,E2 -3710.404} C_VEL
LIN {X 0,Y 546.386,Z 169.224,A -85,B 0,C 180,E1 -3710.658,E2 -3710.658} C_VEL
LIN {X 0,Y 546.909,Z 145.349,A -85,B 0,C 180,E1 -3713.652,E2 -3713.652} C_VEL
LIN {X 0,Y 547.232,Z 127.847,A -85,B 0,C 180,E1 -3715.891,E2 -3715.891} C_VEL
LIN {X 0,Y 545.096,Z 118.213,A -85,B 0,C 180,E1 -3717.272,E2 -3717.272} C_VEL
LIN {X 0,Y 545.079,Z 118.216,A -85,B 0,C 180,E1 -3720.247,E2 -3720.247} C_VEL
LIN {X 0,Y 545.081,Z 118.21,A -85,B 0,C 180,E1 -3723.063,E2 -3723.063} C_VEL
LIN {X 0,Y 545.036,Z 118.222,A -85,B 0,C 180,E1 -3725.673,E2 -3725.673} C_VEL
LIN {X 0,Y 545.055,Z 118.215,A -85,B 0,C 180,E1 -3728.238,E2 -3728.238} C_VEL
LIN {X 0,Y 545.084,Z 118.209,A -85,B 0,C 180,E1 -3730.473,E2 -3730.473} C_VEL
LIN {X 0,Y 545.047,Z 118.214,A -85,B 0,C 180,E1 -3733.11,E2 -3733.11} C_VEL
LIN {X 0,Y 545.052,Z 118.214,A -85,B 0,C 180,E1 -3736.227,E2 -3736.227} C_VEL
LIN {X 0,Y 545.083,Z 118.21,A -85,B 0,C 180,E1 -3738.886,E2 -3738.886} C_VEL
LIN {X 0,Y 545.05,Z 118.214,A -85,B 0,C 180,E1 -3741.865,E2 -3741.865} C_VEL
LIN {X 0,Y 545.039,Z 118.213,A -85,B 0,C 180,E1 -3744.532,E2 -3744.532} C_VEL
LIN {X 0,Y 545.067,Z 118.217,A -85,B 0,C 180,E1 -3747.212,E2 -3747.212} C_VEL
LIN {X 0,Y 545.065,Z 118.21,A -85,B 0,C 180,E1 -3749.811,E2 -3749.811} C_VEL
LIN {X 0,Y 545.062,Z 118.21,A -85,B 0,C 180,E1 -3752.834,E2 -3752.834} C_VEL
LIN {X 0,Y 545.024,Z 118.215,A -85,B 0,C 180,E1 -3755.63,E2 -3755.63} C_VEL
LIN {X 0,Y 545.069,Z 118.208,A -85,B 0,C 180,E1 -3758.181,E2 -3758.181} C_VEL
LIN {X 0,Y 545.12,Z 118.206,A -85,B 0,C 180,E1 -3760.415,E2 -3760.415} C_VEL
LIN {X 0,Y 545.047,Z 118.211,A -85,B 0,C 180,E1 -3763.521,E2 -3763.521} C_VEL
LIN {X 0,Y 545.07,Z 118.209,A -85,B 0,C 180,E1 -3765.82,E2 -3765.82} C_VEL
LIN {X 0,Y 545.121,Z 118.207,A -85,B 0,C 180,E1 -3768.85,E2 -3768.85} C_VEL
LIN {X 0,Y 545.092,Z 118.207,A -85,B 0,C 180,E1 -3771.847,E2 -3771.847} C_VEL
LIN {X 0,Y 545.168,Z 118.199,A -85,B 0,C 180,E1 -3774.823,E2 -3774.823} C_VEL
LIN {X 0,Y 545.193,Z 118.194,A -85,B 0,C 180,E1 -3777.784,E2 -3777.784} C_VEL
LIN {X 0,Y 545.195,Z 118.192,A -85,B 0,C 180,E1 -3780,E2 -3780} C_VEL
LIN {X 0,Y 545.146,Z 118.199,A -85,B 0,C 180,E1 -3782.956,E2 -3782.956} C_VEL
LIN {X 0,Y 545.127,Z 118.209,A -85,B 0,C 180,E1 -3785.92,E2 -3785.92} C_VEL
LIN {X 0,Y 545.07,Z 118.202,A -85,B 0,C 180,E1 -3788.901,E2 -3788.901} C_VEL
LIN {X 0,Y 545.066,Z 118.216,A -85,B 0,C 180,E1 -3791.906,E2 -3791.906} C_VEL
LIN {X 0,Y 545.043,Z 118.212,A -85,B 0,C 180,E1 -3794.945,E2 -3794.945} C_VEL
LIN {X 0,Y 545.035,Z 118.216,A -85,B 0,C 180,E1 -3798.028,E2 -3798.028} C_VEL
LIN {X 0,Y 545.001,Z 118.217,A -85,B 0,C 180,E1 -3800.376,E2 -3800.376} C_VEL
LIN {X 0,Y 544.987,Z 118.218,A -85,B 0,C 180,E1 -3802.76,E2 -3802.76} C_VEL
LIN {X 0,Y 545.014,Z 118.223,A -85,B 0,C 180,E1 -3805.489,E2 -3805.489} C_VEL
LIN {X 0,Y 545,Z 118.217,A -85,B 0,C 180,E1 -3807.661,E2 -3807.661} C_VEL
LIN {X 0,Y 545.025,Z 118.209,A -85,B 0,C 180,E1 -3810.236,E2 -3810.236} C_VEL
LIN {X 0,Y 545.062,Z 118.216,A -85,B 0,C 180,E1 -3813.058,E2 -3813.058} C_VEL
LIN {X 0,Y 545.019,Z 118.215,A -85,B 0,C 180,E1 -3815.67,E2 -3815.67} C_VEL
LIN {X 0,Y 545.004,Z 118.222,A -85,B 0,C 180,E1 -3816.963,E2 -3816.963} C_VEL
LIN {X 0,Y 544.341,Z 118.297,A -85,B 0,C 180,E1 -3817.58,E2 -3817.58} C_VEL
LIN {X 0,Y 541.496,Z 118.651,A -85,B 0,C 180,E1 -3818.582,E2 -3818.582} C_VEL
LIN {X 0,Y 539.093,Z 118.954,A -85,B 0,C 180,E1 -3819.388,E2 -3819.388} C_VEL
LIN {X 0,Y 538.066,Z 119.079,A -85,B 0,C 180,E1 -3820.01,E2 -3820.01} C_VEL
LIN {X 0,Y 537.985,Z 119.09,A -85,B 0,C 180,E1 -3820.221,E2 -3820.221} C_VEL
LIN {X 0,Y 537.975,Z 119.099,A -85,B 0,C 180,E1 -3822.981,E2 -3822.981} C_VEL
LIN {X 0,Y 538.006,Z 119.083,A -85,B 0,C 180,E1 -3825.929,E2 -3825.929} C_VEL
LIN {X 0,Y 537.999,Z 119.091,A -85,B 0,C 180,E1 -3829.26,E2 -3829.26} C_VEL
LIN {X 0,Y 537.99,Z 119.091,A -85,B 0,C 180,E1 -3832.121,E2 -3832.121} C_VEL
LIN {X 0,Y 537.992,Z 119.094,A -85,B 0,C 180,E1 -3834.915,E2 -3834.915} C_VEL
LIN {X 0,Y 538.02,Z 119.085,A -85,B 0,C 180,E1 -3837.617,E2 -3837.617} C_VEL
LIN {X 0,Y 538.005,Z 119.098,A -85,B 0,C 180,E1 -3840.238,E2 -3840.238} C_VEL
LIN {X 0,Y 538.014,Z 119.091,A -85,B 0,C 180,E1 -3842.793,E2 -3842.793} C_VEL
LIN {X 0,Y 537.988,Z 119.092,A -85,B 0,C 180,E1 -3845.289,E2 -3845.289} C_VEL
LIN {X 0,Y 538.021,Z 119.096,A -85,B 0,C 180,E1 -3848.042,E2 -3848.042} C_VEL
LIN {X 0,Y 538.087,Z 119.085,A -85,B 0,C 180,E1 -3850.148,E2 -3850.148} C_VEL
LIN {X 0,Y 537.992,Z 119.09,A -85,B 0,C 180,E1 -3853.298,E2 -3853.298} C_VEL
LIN {X 0,Y 538.057,Z 119.089,A -85,B 0,C 180,E1 -3855.63,E2 -3855.63} C_VEL
LIN {X 0,Y 538.083,Z 119.081,A -85,B 0,C 180,E1 -3858.701,E2 -3858.701} C_VEL
LIN {X 0,Y 538.064,Z 119.09,A -85,B 0,C 180,E1 -3861.739,E2 -3861.739} C_VEL
LIN {X 0,Y 538.172,Z 119.125,A -85,B 0,C 180,E1 -3864.661,E2 -3864.661} C_VEL
LIN {X 0,Y 539.75,Z 127.918,A -85,B 0,C 180,E1 -3866.08,E2 -3866.08} C_VEL
LIN {X 0,Y 539.416,Z 141.739,A -85,B 0,C 180,E1 -3868.133,E2 -3868.133} C_VEL
LIN {X 0,Y 541.839,Z 152.549,A -85,B 0,C 180,E1 -3868.385,E2 -3868.385} C_VEL
LIN {X 0,Y 541.015,Z 306.919,A -85,B 0,C 180,E1 -3870.511,E2 -3870.511} C_VEL
LIN {X 0,Y 540.801,Z 322.531,A -85,B 0,C 180,E1 -3870.884,E2 -3870.884} C_VEL
LIN {X 0,Y 540.468,Z 337.45,A -85,B 0,C 180,E1 -3871.397,E2 -3871.397} C_VEL
LIN {X 0,Y 540.089,Z 351.804,A -85,B 0,C 180,E1 -3872.05,E2 -3872.05} C_VEL
LIN {X 0,Y 539.662,Z 366.338,A -85,B 0,C 180,E1 -3872.892,E2 -3872.892} C_VEL
LIN {X 0,Y 539.304,Z 379.435,A -85,B 0,C 180,E1 -3873.829,E2 -3873.829} C_VEL
LIN {X 0,Y 538.888,Z 391.445,A -85,B 0,C 180,E1 -3874.863,E2 -3874.863} C_VEL
LIN {X 0,Y 538.588,Z 402.417,A -85,B 0,C 180,E1 -3875.992,E2 -3875.992} C_VEL
LIN {X 0,Y 538.259,Z 413.14,A -85,B 0,C 180,E1 -3877.309,E2 -3877.309} C_VEL
LIN {X 0,Y 537.974,Z 422.148,A -85,B 0,C 180,E1 -3878.64,E2 -3878.64} C_VEL
LIN {X 0,Y 537.793,Z 430.612,A -85,B 0,C 180,E1 -3880.161,E2 -3880.161} C_VEL
LIN {X 0,Y 537.658,Z 437.448,A -85,B 0,C 180,E1 -3881.689,E2 -3881.689} C_VEL
LIN {X 0,Y 537.564,Z 442.833,A -85,B 0,C 180,E1 -3883.226,E2 -3883.226} C_VEL
LIN {X 0,Y 537.505,Z 446.523,A -85,B 0,C 180,E1 -3884.63,E2 -3884.63} C_VEL
LIN {X 0,Y 537.443,Z 449.03,A -85,B 0,C 180,E1 -3885.939,E2 -3885.939} C_VEL
LIN {X 0,Y 537.487,Z 450.877,A -85,B 0,C 180,E1 -3887.502,E2 -3887.502} C_VEL
LIN {X 0,Y 537.482,Z 451.498,A -85,B 0,C 180,E1 -3889.08,E2 -3889.08} C_VEL
LIN {X 0,Y 537.444,Z 450.824,A -85,B 0,C 180,E1 -3890.675,E2 -3890.675} C_VEL
LIN {X 0,Y 537.464,Z 448.838,A -85,B 0,C 180,E1 -3892.285,E2 -3892.285} C_VEL
LIN {X 0,Y 537.53,Z 445.462,A -85,B 0,C 180,E1 -3893.911,E2 -3893.911} C_VEL
LIN {X 0,Y 537.601,Z 440.518,A -85,B 0,C 180,E1 -3895.573,E2 -3895.573} C_VEL
LIN {X 0,Y 537.679,Z 435.76,A -85,B 0,C 180,E1 -3896.804,E2 -3896.804} C_VEL
LIN {X 0,Y 537.86,Z 428.825,A -85,B 0,C 180,E1 -3898.272,E2 -3898.272} C_VEL
LIN {X 0,Y 538.052,Z 420.168,A -85,B 0,C 180,E1 -3899.759,E2 -3899.759} C_VEL
LIN {X 0,Y 538.281,Z 411.115,A -85,B 0,C 180,E1 -3901.046,E2 -3901.046} C_VEL
LIN {X 0,Y 538.593,Z 401.231,A -85,B 0,C 180,E1 -3902.229,E2 -3902.229} C_VEL
LIN {X 0,Y 538.917,Z 390.208,A -85,B 0,C 180,E1 -3903.342,E2 -3903.342} C_VEL
LIN {X 0,Y 539.284,Z 378.887,A -85,B 0,C 180,E1 -3904.308,E2 -3904.308} C_VEL
LIN {X 0,Y 539.709,Z 364.782,A -85,B 0,C 180,E1 -3905.299,E2 -3905.299} C_VEL
LIN {X 0,Y 540.159,Z 350.472,A -85,B 0,C 180,E1 -3906.106,E2 -3906.106} C_VEL
LIN {X 0,Y 540.46,Z 336.314,A -85,B 0,C 180,E1 -3906.739,E2 -3906.739} C_VEL
LIN {X 0,Y 540.792,Z 320.942,A -85,B 0,C 180,E1 -3907.251,E2 -3907.251} C_VEL
LIN {X 0,Y 540.995,Z 306.664,A -85,B 0,C 180,E1 -3907.585,E2 -3907.585} C_VEL
LIN {X 0,Y 541.862,Z 152.915,A -85,B 0,C 180,E1 -3909.7,E2 -3909.7} C_VEL
LIN {X 0,Y 539.417,Z 141.773,A -85,B 0,C 180,E1 -3909.971,E2 -3909.971} C_VEL
LIN {X 0,Y 539.795,Z 127.577,A -85,B 0,C 180,E1 -3912.086,E2 -3912.086} C_VEL
LIN {X 0,Y 538.014,Z 119.094,A -85,B 0,C 180,E1 -3913.482,E2 -3913.482} C_VEL
LIN {X 0,Y 538.005,Z 119.097,A -85,B 0,C 180,E1 -3916.184,E2 -3916.184} C_VEL
LIN {X 0,Y 538.025,Z 119.091,A -85,B 0,C 180,E1 -3919.256,E2 -3919.256} C_VEL
LIN {X 0,Y 537.99,Z 119.1,A -85,B 0,C 180,E1 -3922.121,E2 -3922.121} C_VEL
LIN {X 0,Y 537.996,Z 119.09,A -85,B 0,C 180,E1 -3924.915,E2 -3924.915} C_VEL
LIN {X 0,Y 538.02,Z 119.089,A -85,B 0,C 180,E1 -3927.617,E2 -3927.617} C_VEL
LIN {X 0,Y 538.011,Z 119.095,A -85,B 0,C 180,E1 -3930.238,E2 -3930.238} C_VEL
LIN {X 0,Y 538.035,Z 119.086,A -85,B 0,C 180,E1 -3932.794,E2 -3932.794} C_VEL
LIN {X 0,Y 537.996,Z 119.09,A -85,B 0,C 180,E1 -3935.29,E2 -3935.29} C_VEL
LIN {X 0,Y 538.017,Z 119.096,A -85,B 0,C 180,E1 -3938.042,E2 -3938.042} C_VEL
LIN {X 0,Y 538.082,Z 119.085,A -85,B 0,C 180,E1 -3940.148,E2 -3940.148} C_VEL
LIN {X 0,Y 537.997,Z 119.092,A -85,B 0,C 180,E1 -3943.298,E2 -3943.298} C_VEL
LIN {X 0,Y 538.053,Z 119.089,A -85,B 0,C 180,E1 -3945.63,E2 -3945.63} C_VEL
LIN {X 0,Y 538.079,Z 119.079,A -85,B 0,C 180,E1 -3948.701,E2 -3948.701} C_VEL
LIN {X 0,Y 538.083,Z 119.087,A -85,B 0,C 180,E1 -3951.739,E2 -3951.739} C_VEL
LIN {X 0,Y 538.16,Z 119.068,A -85,B 0,C 180,E1 -3954.755,E2 -3954.755} C_VEL
LIN {X 0,Y 538.171,Z 119.072,A -85,B 0,C 180,E1 -3957.754,E2 -3957.754} C_VEL
LIN {X 0,Y 538.179,Z 119.069,A -85,B 0,C 180,E1 -3960.748,E2 -3960.748} C_VEL
LIN {X 0,Y 538.134,Z 119.077,A -85,B 0,C 180,E1 -3962.994,E2 -3962.994} C_VEL
LIN {X 0,Y 538.121,Z 119.075,A -85,B 0,C 180,E1 -3965.997,E2 -3965.997} C_VEL
LIN {X 0,Y 538.055,Z 119.089,A -85,B 0,C 180,E1 -3969.018,E2 -3969.018} C_VEL
LIN {X 0,Y 538.083,Z 119.078,A -85,B 0,C 180,E1 -3972.062,E2 -3972.062} C_VEL
LIN {X 0,Y 538.045,Z 119.089,A -85,B 0,C 180,E1 -3975.144,E2 -3975.144} C_VEL
LIN {X 0,Y 538.024,Z 119.088,A -85,B 0,C 180,E1 -3978.27,E2 -3978.27} C_VEL
LIN {X 0,Y 538.037,Z 119.089,A -85,B 0,C 180,E1 -3980.651,E2 -3980.651} C_VEL
LIN {X 0,Y 538.003,Z 119.089,A -85,B 0,C 180,E1 -3983.888,E2 -3983.888} C_VEL
LIN {X 0,Y 538.041,Z 119.088,A -85,B 0,C 180,E1 -3986.366,E2 -3986.366} C_VEL
LIN {X 0,Y 538.029,Z 119.09,A -85,B 0,C 180,E1 -3988.933,E2 -3988.933} C_VEL
LIN {X 0,Y 538.009,Z 119.089,A -85,B 0,C 180,E1 -3991.887,E2 -3991.887} C_VEL
LIN {X 0,Y 538.008,Z 119.095,A -85,B 0,C 180,E1 -3994.617,E2 -3994.617} C_VEL
LIN {X 0,Y 538.003,Z 119.089,A -85,B 0,C 180,E1 -3997.17,E2 -3997.17} C_VEL
LIN {X 0,Y 538.021,Z 119.086,A -85,B 0,C 180,E1 -3999.797,E2 -3999.797} C_VEL
LIN {X 0,Y 538.017,Z 119.087,A -85,B 0,C 180,E1 -4002.786,E2 -4002.786} C_VEL
LIN {X 0,Y 538.031,Z 119.087,A -85,B 0,C 180,E1 -4005.141,E2 -4005.141} C_VEL
LIN {X 0,Y 538.029,Z 119.095,A -85,B 0,C 180,E1 -4008.227,E2 -4008.227} C_VEL
LIN {X 0,Y 538.015,Z 119.089,A -85,B 0,C 180,E1 -4011.17,E2 -4011.17} C_VEL
LIN {X 0,Y 537.993,Z 119.099,A -85,B 0,C 180,E1 -4014.089,E2 -4014.089} C_VEL
LIN {X 0,Y 538.029,Z 119.087,A -85,B 0,C 180,E1 -4016.728,E2 -4016.728} C_VEL
LIN {X 0,Y 538.025,Z 119.093,A -85,B 0,C 180,E1 -4019.556,E2 -4019.556} C_VEL
LIN {X 0,Y 538.054,Z 119.091,A -85,B 0,C 180,E1 -4022.505,E2 -4022.505} C_VEL
LIN {X 0,Y 540.384,Z 129.491,A -85,B 0,C 180,E1 -4024.014,E2 -4024.014} C_VEL
LIN {X 0,Y 539.93,Z 149.581,A -85,B 0,C 180,E1 -4026.609,E2 -4026.609} C_VEL
LIN {X 0,Y 539.468,Z 169.025,A -85,B 0,C 180,E1 -4029.077,E2 -4029.077} C_VEL
LIN {X 0,Y 541.809,Z 181.604,A -85,B 0,C 180,E1 -4029.348,E2 -4029.348} C_VEL
LIN {X 0,Y 540.942,Z 335.589,A -85,B 0,C 180,E1 -4031.462,E2 -4031.462} C_VEL
LIN {X 0,Y 540.715,Z 350.9,A -85,B 0,C 180,E1 -4031.824,E2 -4031.824} C_VEL
LIN {X 0,Y 540.459,Z 365.08,A -85,B 0,C 180,E1 -4032.304,E2 -4032.304} C_VEL
LIN {X 0,Y 540.064,Z 378.156,A -85,B 0,C 180,E1 -4032.877,E2 -4032.877} C_VEL
LIN {X 0,Y 539.672,Z 392.113,A -85,B 0,C 180,E1 -4033.644,E2 -4033.644} C_VEL
LIN {X 0,Y 539.325,Z 404.596,A -85,B 0,C 180,E1 -4034.484,E2 -4034.484} C_VEL
LIN {X 0,Y 538.894,Z 417.818,A -85,B 0,C 180,E1 -4035.557,E2 -4035.557} C_VEL
LIN {X 0,Y 538.591,Z 428.639,A -85,B 0,C 180,E1 -4036.608,E2 -4036.608} C_VEL
LIN {X 0,Y 538.291,Z 438.649,A -85,B 0,C 180,E1 -4037.751,E2 -4037.751} C_VEL
LIN {X 0,Y 538.073,Z 448.441,A -85,B 0,C 180,E1 -4039.083,E2 -4039.083} C_VEL
LIN {X 0,Y 537.824,Z 456.608,A -85,B 0,C 180,E1 -4040.409,E2 -4040.409} C_VEL
LIN {X 0,Y 537.733,Z 463.36,A -85,B 0,C 180,E1 -4041.734,E2 -4041.734} C_VEL
LIN {X 0,Y 537.618,Z 469.594,A -85,B 0,C 180,E1 -4043.244,E2 -4043.244} C_VEL
LIN {X 0,Y 537.574,Z 474.386,A -85,B 0,C 180,E1 -4044.75,E2 -4044.75} C_VEL
LIN {X 0,Y 537.561,Z 477.887,A -85,B 0,C 180,E1 -4046.252,E2 -4046.252} C_VEL
LIN {X 0,Y 537.487,Z 480.189,A -85,B 0,C 180,E1 -4047.752,E2 -4047.752} C_VEL
LIN {X 0,Y 537.438,Z 481.347,A -85,B 0,C 180,E1 -4049.251,E2 -4049.251} C_VEL
LIN {X 0,Y 537.438,Z 481.346,A -85,B 0,C 180,E1 -4050.75,E2 -4050.75} C_VEL
LIN {X 0,Y 537.488,Z 480.184,A -85,B 0,C 180,E1 -4052.248,E2 -4052.248} C_VEL
LIN {X 0,Y 537.562,Z 477.881,A -85,B 0,C 180,E1 -4053.748,E2 -4053.748} C_VEL
LIN {X 0,Y 537.574,Z 474.385,A -85,B 0,C 180,E1 -4055.251,E2 -4055.251} C_VEL
LIN {X 0,Y 537.664,Z 469.597,A -85,B 0,C 180,E1 -4056.756,E2 -4056.756} C_VEL
LIN {X 0,Y 537.733,Z 463.356,A -85,B 0,C 180,E1 -4058.266,E2 -4058.266} C_VEL
LIN {X 0,Y 537.855,Z 455.516,A -85,B 0,C 180,E1 -4059.78,E2 -4059.78} C_VEL
LIN {X 0,Y 538.081,Z 447.18,A -85,B 0,C 180,E1 -4061.108,E2 -4061.108} C_VEL
LIN {X 0,Y 538.33,Z 437.134,A -85,B 0,C 180,E1 -4062.44,E2 -4062.44} C_VEL
LIN {X 0,Y 538.631,Z 426.86,A -85,B 0,C 180,E1 -4063.584,E2 -4063.584} C_VEL
LIN {X 0,Y 539.002,Z 414.619,A -85,B 0,C 180,E1 -4064.73,E2 -4064.73} C_VEL
LIN {X 0,Y 539.442,Z 401.04,A -85,B 0,C 180,E1 -4065.778,E2 -4065.778} C_VEL
LIN {X 0,Y 539.871,Z 387.325,A -85,B 0,C 180,E1 -4066.643,E2 -4066.643} C_VEL
LIN {X 0,Y 540.209,Z 373.168,A -85,B 0,C 180,E1 -4067.363,E2 -4067.363} C_VEL
LIN {X 0,Y 540.581,Z 357.859,A -85,B 0,C 180,E1 -4067.961,E2 -4067.961} C_VEL
LIN {X 0,Y 540.857,Z 343.087,A -85,B 0,C 180,E1 -4068.381,E2 -4068.381} C_VEL
LIN {X 0,Y 541.05,Z 327.334,A -85,B 0,C 180,E1 -4068.669,E2 -4068.669} C_VEL
LIN {X 0,Y 541.741,Z 180.812,A -85,B 0,C 180,E1 -4070.667,E2 -4070.667} C_VEL
LIN {X 0,Y 539.478,Z 169.027,A -85,B 0,C 180,E1 -4070.935,E2 -4070.935} C_VEL
LIN {X 0,Y 540.006,Z 148.114,A -85,B 0,C 180,E1 -4073.591,E2 -4073.591} C_VEL
LIN {X 0,Y 540.431,Z 129.54,A -85,B 0,C 180,E1 -4075.996,E2 -4075.996} C_VEL
LIN {X 0,Y 538.048,Z 119.091,A -85,B 0,C 180,E1 -4077.518,E2 -4077.518} C_VEL
LIN {X 0,Y 538.022,Z 119.091,A -85,B 0,C 180,E1 -4080.627,E2 -4080.627} C_VEL
LIN {X 0,Y 538.048,Z 119.087,A -85,B 0,C 180,E1 -4083.283,E2 -4083.283} C_VEL
LIN {X 0,Y 537.996,Z 119.099,A -85,B 0,C 180,E1 -4086.005,E2 -4086.005} C_VEL
LIN {X 0,Y 538.017,Z 119.088,A -85,B 0,C 180,E1 -4088.831,E2 -4088.831} C_VEL
LIN {X 0,Y 538.026,Z 119.095,A -85,B 0,C 180,E1 -4091.774,E2 -4091.774} C_VEL
LIN {X 0,Y 538.009,Z 119.09,A -85,B 0,C 180,E1 -4094.863,E2 -4094.863} C_VEL
LIN {X 0,Y 538.021,Z 119.093,A -85,B 0,C 180,E1 -4097.214,E2 -4097.214} C_VEL
LIN {X 0,Y 538.013,Z 119.088,A -85,B 0,C 180,E1 -4100.202,E2 -4100.202} C_VEL
LIN {X 0,Y 538.027,Z 119.091,A -85,B 0,C 180,E1 -4103.067,E2 -4103.067} C_VEL
LIN {X 0,Y 538.013,Z 119.09,A -85,B 0,C 180,E1 -4105.827,E2 -4105.827} C_VEL
LIN {X 0,Y 538.011,Z 119.089,A -85,B 0,C 180,E1 -4108.499,E2 -4108.499} C_VEL
LIN {X 0,Y 538.022,Z 119.091,A -85,B 0,C 180,E1 -4111.098,E2 -4111.098} C_VEL
LIN {X 0,Y 538.035,Z 119.084,A -85,B 0,C 180,E1 -4113.633,E2 -4113.633} C_VEL
LIN {X 0,Y 538.01,Z 119.096,A -85,B 0,C 180,E1 -4116.928,E2 -4116.928} C_VEL
LIN {X 0,Y 538.085,Z 119.079,A -85,B 0,C 180,E1 -4120.148,E2 -4120.148} C_VEL
LIN {X 0,Y 537.998,Z 119.09,A -85,B 0,C 180,E1 -4123.298,E2 -4123.298} C_VEL
LIN {X 0,Y 538.043,Z 119.084,A -85,B 0,C 180,E1 -4125.63,E2 -4125.63} C_VEL
LIN {X 0,Y 538.081,Z 119.086,A -85,B 0,C 180,E1 -4128.702,E2 -4128.702} C_VEL
LIN {X 0,Y 538.057,Z 119.082,A -85,B 0,C 180,E1 -4131.739,E2 -4131.739} C_VEL
LIN {X 0,Y 538.127,Z 119.077,A -85,B 0,C 180,E1 -4134.755,E2 -4134.755} C_VEL
LIN {X 0,Y 538.165,Z 119.069,A -85,B 0,C 180,E1 -4137.755,E2 -4137.755} C_VEL
LIN {X 0,Y 538.163,Z 119.067,A -85,B 0,C 180,E1 -4140,E2 -4140} C_VEL
LIN {X 0,Y 538.114,Z 119.074,A -85,B 0,C 180,E1 -4142.995,E2 -4142.995} C_VEL
LIN {X 0,Y 538.083,Z 119.086,A -85,B 0,C 180,E1 -4145.998,E2 -4145.998} C_VEL
LIN {X 0,Y 538.028,Z 119.079,A -85,B 0,C 180,E1 -4149.019,E2 -4149.019} C_VEL
LIN {X 0,Y 538.018,Z 119.091,A -85,B 0,C 180,E1 -4152.064,E2 -4152.064} C_VEL
LIN {X 0,Y 537.991,Z 119.092,A -85,B 0,C 180,E1 -4155.146,E2 -4155.146} C_VEL
LIN {X 0,Y 537.984,Z 119.092,A -85,B 0,C 180,E1 -4158.272,E2 -4158.272} C_VEL
LIN {X 0,Y 537.97,Z 119.093,A -85,B 0,C 180,E1 -4160.655,E2 -4160.655} C_VEL
LIN {X 0,Y 537.976,Z 119.094,A -85,B 0,C 180,E1 -4163.074,E2 -4163.074} C_VEL
LIN {X 0,Y 537.975,Z 119.097,A -85,B 0,C 180,E1 -4165.656,E2 -4165.656} C_VEL
LIN {X 0,Y 537.974,Z 119.088,A -85,B 0,C 180,E1 -4168.054,E2 -4168.054} C_VEL
LIN {X 0,Y 537.992,Z 119.086,A -85,B 0,C 180,E1 -4170.629,E2 -4170.629} C_VEL
LIN {X 0,Y 538.004,Z 119.096,A -85,B 0,C 180,E1 -4173.275,E2 -4173.275} C_VEL
LIN {X 0,Y 537.958,Z 119.093,A -85,B 0,C 180,E1 -4176.008,E2 -4176.008} C_VEL
LIN {X 0,Y 537.993,Z 119.09,A -85,B 0,C 180,E1 -4178.833,E2 -4178.833} C_VEL
LIN {X 0,Y 537.985,Z 119.09,A -85,B 0,C 180,E1 -4180.221,E2 -4180.221} C_VEL
LIN {X 0,Y 537.324,Z 119.179,A -85,B 0,C 180,E1 -4180.846,E2 -4180.846} C_VEL
LIN {X 0,Y 534.472,Z 119.534,A -85,B 0,C 180,E1 -4181.861,E2 -4181.861} C_VEL
LIN {X 0,Y 532.055,Z 119.836,A -85,B 0,C 180,E1 -4182.678,E2 -4182.678} C_VEL
LIN {X 0,Y 531.015,Z 119.961,A -85,B 0,C 180,E1 -4183.308,E2 -4183.308} C_VEL
LIN {X 0,Y 530.93,Z 119.97,A -85,B 0,C 180,E1 -4183.522,E2 -4183.522} C_VEL
LIN {X 0,Y 530.97,Z 119.959,A -85,B 0,C 180,E1 -4185.623,E2 -4185.623} C_VEL
LIN {X 0,Y 530.936,Z 119.974,A -85,B 0,C 180,E1 -4188.983,E2 -4188.983} C_VEL
LIN {X 0,Y 530.954,Z 119.965,A -85,B 0,C 180,E1 -4191.528,E2 -4191.528} C_VEL
LIN {X 0,Y 530.952,Z 119.974,A -85,B 0,C 180,E1 -4194.379,E2 -4194.379} C_VEL
LIN {X 0,Y 530.971,Z 119.963,A -85,B 0,C 180,E1 -4197.133,E2 -4197.133} C_VEL
LIN {X 0,Y 530.956,Z 119.97,A -85,B 0,C 180,E1 -4199.802,E2 -4199.802} C_VEL
LIN {X 0,Y 530.968,Z 119.972,A -85,B 0,C 180,E1 -4202.478,E2 -4202.478} C_VEL
LIN {X 0,Y 530.955,Z 119.969,A -85,B 0,C 180,E1 -4204.939,E2 -4204.939} C_VEL
LIN {X 0,Y 530.982,Z 119.971,A -85,B 0,C 180,E1 -4207.898,E2 -4207.898} C_VEL
LIN {X 0,Y 530.986,Z 119.964,A -85,B 0,C 180,E1 -4210.677,E2 -4210.677} C_VEL
LIN {X 0,Y 530.959,Z 119.965,A -85,B 0,C 180,E1 -4213.07,E2 -4213.07} C_VEL
LIN {X 0,Y 531.014,Z 119.964,A -85,B 0,C 180,E1 -4215.435,E2 -4215.435} C_VEL
LIN {X 0,Y 531.041,Z 119.959,A -85,B 0,C 180,E1 -4218.549,E2 -4218.549} C_VEL
LIN {X 0,Y 531.039,Z 119.966,A -85,B 0,C 180,E1 -4221.629,E2 -4221.629} C_VEL
LIN {X 0,Y 531.135,Z 120.124,A -85,B 0,C 180,E1 -4224.447,E2 -4224.447} C_VEL
LIN {X 0,Y 532.869,Z 128.583,A -85,B 0,C 180,E1 -4225.84,E2 -4225.84} C_VEL
LIN {X 0,Y 532.603,Z 141.912,A -85,B 0,C 180,E1 -4227.849,E2 -4227.849} C_VEL
LIN {X 0,Y 535.102,Z 153.073,A -85,B 0,C 180,E1 -4228.118,E2 -4228.118} C_VEL
LIN {X 0,Y 534.483,Z 281.994,A -85,B 0,C 180,E1 -4229.906,E2 -4229.906} C_VEL
LIN {X 0,Y 534.273,Z 308.314,A -85,B 0,C 180,E1 -4230.296,E2 -4230.296} C_VEL
LIN {X 0,Y 534.019,Z 323.61,A -85,B 0,C 180,E1 -4230.676,E2 -4230.676} C_VEL
LIN {X 0,Y 533.691,Z 337.907,A -85,B 0,C 180,E1 -4231.179,E2 -4231.179} C_VEL
LIN {X 0,Y 533.324,Z 351.274,A -85,B 0,C 180,E1 -4231.793,E2 -4231.793} C_VEL
LIN {X 0,Y 532.838,Z 366.005,A -85,B 0,C 180,E1 -4232.646,E2 -4232.646} C_VEL
LIN {X 0,Y 532.376,Z 379.227,A -85,B 0,C 180,E1 -4233.595,E2 -4233.595} C_VEL
LIN {X 0,Y 531.965,Z 390.248,A -85,B 0,C 180,E1 -4234.546,E2 -4234.546} C_VEL
LIN {X 0,Y 531.655,Z 401.42,A -85,B 0,C 180,E1 -4235.69,E2 -4235.69} C_VEL
LIN {X 0,Y 531.309,Z 411.665,A -85,B 0,C 180,E1 -4236.935,E2 -4236.935} C_VEL
LIN {X 0,Y 531.009,Z 420.288,A -85,B 0,C 180,E1 -4238.179,E2 -4238.179} C_VEL
LIN {X 0,Y 530.795,Z 428.127,A -85,B 0,C 180,E1 -4239.526,E2 -4239.526} C_VEL
LIN {X 0,Y 530.624,Z 435.406,A -85,B 0,C 180,E1 -4241.053,E2 -4241.053} C_VEL
LIN {X 0,Y 530.508,Z 441.344,A -85,B 0,C 180,E1 -4242.626,E2 -4242.626} C_VEL
LIN {X 0,Y 530.465,Z 444.832,A -85,B 0,C 180,E1 -4243.796,E2 -4243.796} C_VEL
LIN {X 0,Y 530.369,Z 448.331,A -85,B 0,C 180,E1 -4245.368,E2 -4245.368} C_VEL
LIN {X 0,Y 530.364,Z 450.575,A -85,B 0,C 180,E1 -4246.949,E2 -4246.949} C_VEL
LIN {X 0,Y 530.368,Z 451.591,A -85,B 0,C 180,E1 -4248.543,E2 -4248.543} C_VEL
LIN {X 0,Y 530.35,Z 451.361,A -85,B 0,C 180,E1 -4250.154,E2 -4250.154} C_VEL
LIN {X 0,Y 530.41,Z 449.841,A -85,B 0,C 180,E1 -4251.777,E2 -4251.777} C_VEL
LIN {X 0,Y 530.442,Z 446.954,A -85,B 0,C 180,E1 -4253.42,E2 -4253.42} C_VEL
LIN {X 0,Y 530.495,Z 442.579,A -85,B 0,C 180,E1 -4255.083,E2 -4255.083} C_VEL
LIN {X 0,Y 530.602,Z 438.234,A -85,B 0,C 180,E1 -4256.341,E2 -4256.341} C_VEL
LIN {X 0,Y 530.677,Z 432.856,A -85,B 0,C 180,E1 -4257.614,E2 -4257.614} C_VEL
LIN {X 0,Y 530.864,Z 425.199,A -85,B 0,C 180,E1 -4259.1,E2 -4259.1} C_VEL
LIN {X 0,Y 531.137,Z 416.87,A -85,B 0,C 180,E1 -4260.434,E2 -4260.434} C_VEL
LIN {X 0,Y 531.458,Z 407.348,A -85,B 0,C 180,E1 -4261.712,E2 -4261.712} C_VEL
LIN {X 0,Y 531.809,Z 396.624,A -85,B 0,C 180,E1 -4262.92,E2 -4262.92} C_VEL
LIN {X 0,Y 532.228,Z 384.919,A -85,B 0,C 180,E1 -4264.025,E2 -4264.025} C_VEL
LIN {X 0,Y 532.692,Z 372.318,A -85,B 0,C 180,E1 -4265.015,E2 -4265.015} C_VEL
LIN {X 0,Y 533.059,Z 360.169,A -85,B 0,C 180,E1 -4265.806,E2 -4265.806} C_VEL
LIN {X 0,Y 533.475,Z 346.701,A -85,B 0,C 180,E1 -4266.523,E2 -4266.523} C_VEL
LIN {X 0,Y 533.793,Z 333.224,A -85,B 0,C 180,E1 -4267.091,E2 -4267.091} C_VEL
LIN {X 0,Y 534.11,Z 318.173,A -85,B 0,C 180,E1 -4267.566,E2 -4267.566} C_VEL
LIN {X 0,Y 534.311,Z 302.986,A -85,B 0,C 180,E1 -4267.888,E2 -4267.888} C_VEL
LIN {X 0,Y 535.212,Z 153.766,A -85,B 0,C 180,E1 -4269.959,E2 -4269.959} C_VEL
LIN {X 0,Y 532.564,Z 142.011,A -85,B 0,C 180,E1 -4270.25,E2 -4270.25} C_VEL
LIN {X 0,Y 532.842,Z 128.613,A -85,B 0,C 180,E1 -4272.273,E2 -4272.273} C_VEL
LIN {X 0,Y 530.999,Z 119.969,A -85,B 0,C 180,E1 -4273.731,E2 -4273.731} C_VEL
LIN {X 0,Y 530.946,Z 119.977,A -85,B 0,C 180,E1 -4276.721,E2 -4276.721} C_VEL
LIN {X 0,Y 530.967,Z 119.971,A -85,B 0,C 180,E1 -4279.565,E2 -4279.565} C_VEL
LIN {X 0,Y 530.967,Z 119.973,A -85,B 0,C 180,E1 -4282.577,E2 -4282.577} C_VEL
LIN {X 0,Y 530.982,Z 119.962,A -85,B 0,C 180,E1 -4285.309,E2 -4285.309} C_VEL
LIN {X 0,Y 530.968,Z 119.97,A -85,B 0,C 180,E1 -4288.031,E2 -4288.031} C_VEL
LIN {X 0,Y 530.989,Z 119.962,A -85,B 0,C 180,E1 -4290.874,E2 -4290.874} C_VEL
LIN {X 0,Y 530.987,Z 119.964,A -85,B 0,C 180,E1 -4293.255,E2 -4293.255} C_VEL
LIN {X 0,Y 530.955,Z 119.97,A -85,B 0,C 180,E1 -4295.968,E2 -4295.968} C_VEL
LIN {X 0,Y 531,Z 119.962,A -85,B 0,C 180,E1 -4299.062,E2 -4299.062} C_VEL
LIN {X 0,Y 530.973,Z 119.969,A -85,B 0,C 180,E1 -4301.478,E2 -4301.478} C_VEL
LIN {X 0,Y 530.991,Z 119.962,A -85,B 0,C 180,E1 -4304.65,E2 -4304.65} C_VEL
LIN {X 0,Y 531.028,Z 119.964,A -85,B 0,C 180,E1 -4307.774,E2 -4307.774} C_VEL
LIN {X 0,Y 530.981,Z 119.966,A -85,B 0,C 180,E1 -4310.092,E2 -4310.092} C_VEL
LIN {X 0,Y 531.072,Z 119.955,A -85,B 0,C 180,E1 -4312.988,E2 -4312.988} C_VEL
LIN {X 0,Y 531.119,Z 119.945,A -85,B 0,C 180,E1 -4314.685,E2 -4314.685} C_VEL
LIN {X 0,Y 531.142,Z 119.947,A -85,B 0,C 180,E1 -4317.725,E2 -4317.725} C_VEL
LIN {X 0,Y 531.15,Z 119.945,A -85,B 0,C 180,E1 -4320.758,E2 -4320.758} C_VEL
LIN {X 0,Y 531.101,Z 119.953,A -85,B 0,C 180,E1 -4323.034,E2 -4323.034} C_VEL
LIN {X 0,Y 531.075,Z 119.952,A -85,B 0,C 180,E1 -4326.077,E2 -4326.077} C_VEL
LIN {X 0,Y 531.017,Z 119.965,A -85,B 0,C 180,E1 -4329.138,E2 -4329.138} C_VEL
LIN {X 0,Y 531.04,Z 119.956,A -85,B 0,C 180,E1 -4332.225,E2 -4332.225} C_VEL
LIN {X 0,Y 530.994,Z 119.964,A -85,B 0,C 180,E1 -4335.35,E2 -4335.35} C_VEL
LIN {X 0,Y 530.984,Z 119.967,A -85,B 0,C 180,E1 -4338.521,E2 -4338.521} C_VEL
LIN {X 0,Y 530.998,Z 119.97,A -85,B 0,C 180,E1 -4340.938,E2 -4340.938} C_VEL
LIN {X 0,Y 530.971,Z 119.967,A -85,B 0,C 180,E1 -4344.225,E2 -4344.225} C_VEL
LIN {X 0,Y 531.001,Z 119.968,A -85,B 0,C 180,E1 -4346.744,E2 -4346.744} C_VEL
LIN {X 0,Y 530.98,Z 119.964,A -85,B 0,C 180,E1 -4349.323,E2 -4349.323} C_VEL
LIN {X 0,Y 530.964,Z 119.968,A -85,B 0,C 180,E1 -4352.1,E2 -4352.1} C_VEL
LIN {X 0,Y 530.967,Z 119.97,A -85,B 0,C 180,E1 -4354.851,E2 -4354.851} C_VEL
LIN {X 0,Y 530.964,Z 119.965,A -85,B 0,C 180,E1 -4357.508,E2 -4357.508} C_VEL
LIN {X 0,Y 530.98,Z 119.973,A -85,B 0,C 180,E1 -4360.433,E2 -4360.433} C_VEL
LIN {X 0,Y 530.964,Z 119.963,A -85,B 0,C 180,E1 -4363.495,E2 -4363.495} C_VEL
LIN {X 0,Y 530.964,Z 119.969,A -85,B 0,C 180,E1 -4366.505,E2 -4366.505} C_VEL
LIN {X 0,Y 530.981,Z 119.966,A -85,B 0,C 180,E1 -4369.567,E2 -4369.567} C_VEL
LIN {X 0,Y 530.967,Z 119.968,A -85,B 0,C 180,E1 -4372.577,E2 -4372.577} C_VEL
LIN {X 0,Y 530.981,Z 119.965,A -85,B 0,C 180,E1 -4375.31,E2 -4375.31} C_VEL
LIN {X 0,Y 530.966,Z 119.974,A -85,B 0,C 180,E1 -4378.032,E2 -4378.032} C_VEL
LIN {X 0,Y 530.988,Z 119.968,A -85,B 0,C 180,E1 -4380.874,E2 -4380.874} C_VEL
LIN {X 0,Y 531.052,Z 120.057,A -85,B 0,C 180,E1 -4382.273,E2 -4382.273} C_VEL
LIN {X 0,Y 533.572,Z 131.493,A -85,B 0,C 180,E1 -4383.947,E2 -4383.947} C_VEL
LIN {X 0,Y 533.038,Z 152.522,A -85,B 0,C 180,E1 -4386.7,E2 -4386.7} C_VEL
LIN {X 0,Y 532.584,Z 168.791,A -85,B 0,C 180,E1 -4388.791,E2 -4388.791} C_VEL
LIN {X 0,Y 535.157,Z 182.149,A -85,B 0,C 180,E1 -4389.09,E2 -4389.09} C_VEL
LIN {X 0,Y 534.221,Z 335.247,A -85,B 0,C 180,E1 -4391.22,E2 -4391.22} C_VEL
LIN {X 0,Y 533.955,Z 350.622,A -85,B 0,C 180,E1 -4391.586,E2 -4391.586} C_VEL
LIN {X 0,Y 533.66,Z 364.816,A -85,B 0,C 180,E1 -4392.071,E2 -4392.071} C_VEL
LIN {X 0,Y 533.231,Z 377.905,A -85,B 0,C 180,E1 -4392.651,E2 -4392.651} C_VEL
LIN {X 0,Y 532.8,Z 391.871,A -85,B 0,C 180,E1 -4393.427,E2 -4393.427} C_VEL
LIN {X 0,Y 532.409,Z 404.666,A -85,B 0,C 180,E1 -4394.3,E2 -4394.3} C_VEL
LIN {X 0,Y 531.951,Z 417.588,A -85,B 0,C 180,E1 -4395.364,E2 -4395.364} C_VEL
LIN {X 0,Y 531.593,Z 428.413,A -85,B 0,C 180,E1 -4396.428,E2 -4396.428} C_VEL
LIN {X 0,Y 531.272,Z 438.427,A -85,B 0,C 180,E1 -4397.587,E2 -4397.587} C_VEL
LIN {X 0,Y 531.001,Z 448.223,A -85,B 0,C 180,E1 -4398.936,E2 -4398.936} C_VEL
LIN {X 0,Y 530.776,Z 456.396,A -85,B 0,C 180,E1 -4400.281,E2 -4400.281} C_VEL
LIN {X 0,Y 530.664,Z 463.149,A -85,B 0,C 180,E1 -4401.624,E2 -4401.624} C_VEL
LIN {X 0,Y 530.549,Z 469.387,A -85,B 0,C 180,E1 -4403.153,E2 -4403.153} C_VEL
LIN {X 0,Y 530.509,Z 474.211,A -85,B 0,C 180,E1 -4404.679,E2 -4404.679} C_VEL
LIN {X 0,Y 530.481,Z 477.745,A -85,B 0,C 180,E1 -4406.202,E2 -4406.202} C_VEL
LIN {X 0,Y 530.408,Z 480.067,A -85,B 0,C 180,E1 -4407.722,E2 -4407.722} C_VEL
LIN {X 0,Y 530.34,Z 481.235,A -85,B 0,C 180,E1 -4409.241,E2 -4409.241} C_VEL
LIN {X 0,Y 530.34,Z 481.234,A -85,B 0,C 180,E1 -4410.76,E2 -4410.76} C_VEL
LIN {X 0,Y 530.409,Z 480.064,A -85,B 0,C 180,E1 -4412.278,E2 -4412.278} C_VEL
LIN {X 0,Y 530.481,Z 477.741,A -85,B 0,C 180,E1 -4413.798,E2 -4413.798} C_VEL
LIN {X 0,Y 530.509,Z 474.215,A -85,B 0,C 180,E1 -4415.321,E2 -4415.321} C_VEL
LIN {X 0,Y 530.569,Z 469.396,A -85,B 0,C 180,E1 -4416.847,E2 -4416.847} C_VEL
LIN {X 0,Y 530.665,Z 463.153,A -85,B 0,C 180,E1 -4418.377,E2 -4418.377} C_VEL
LIN {X 0,Y 530.804,Z 455.311,A -85,B 0,C 180,E1 -4419.912,E2 -4419.912} C_VEL
LIN {X 0,Y 531.024,Z 446.972,A -85,B 0,C 180,E1 -4421.258,E2 -4421.258} C_VEL
LIN {X 0,Y 531.323,Z 436.924,A -85,B 0,C 180,E1 -4422.607,E2 -4422.607} C_VEL
LIN {X 0,Y 531.661,Z 426.648,A -85,B 0,C 180,E1 -4423.765,E2 -4423.765} C_VEL
LIN {X 0,Y 532.056,Z 414.402,A -85,B 0,C 180,E1 -4424.927,E2 -4424.927} C_VEL
LIN {X 0,Y 532.521,Z 402.116,A -85,B 0,C 180,E1 -4425.894,E2 -4425.894} C_VEL
LIN {X 0,Y 532.969,Z 388.737,A -85,B 0,C 180,E1 -4426.766,E2 -4426.766} C_VEL
LIN {X 0,Y 533.372,Z 373.97,A -85,B 0,C 180,E1 -4427.543,E2 -4427.543} C_VEL
LIN {X 0,Y 533.775,Z 359.677,A -85,B 0,C 180,E1 -4428.124,E2 -4428.124} C_VEL
LIN {X 0,Y 534.052,Z 344.715,A -85,B 0,C 180,E1 -4428.574,E2 -4428.574} C_VEL
LIN {X 0,Y 534.297,Z 329.454,A -85,B 0,C 180,E1 -4428.876,E2 -4428.876} C_VEL
LIN {X 0,Y 535.158,Z 182.609,A -85,B 0,C 180,E1 -4430.905,E2 -4430.905} C_VEL
LIN {X 0,Y 532.579,Z 168.891,A -85,B 0,C 180,E1 -4431.211,E2 -4431.211} C_VEL
LIN {X 0,Y 533.138,Z 149.503,A -85,B 0,C 180,E1 -4433.708,E2 -4433.708} C_VEL
LIN {X 0,Y 533.624,Z 131.576,A -85,B 0,C 180,E1 -4436.057,E2 -4436.057} C_VEL
LIN {X 0,Y 530.991,Z 119.971,A -85,B 0,C 180,E1 -4437.758,E2 -4437.758} C_VEL
LIN {X 0,Y 530.976,Z 119.969,A -85,B 0,C 180,E1 -4440.645,E2 -4440.645} C_VEL
LIN {X 0,Y 530.989,Z 119.972,A -85,B 0,C 180,E1 -4443.773,E2 -4443.773} C_VEL
LIN {X 0,Y 530.957,Z 119.97,A -85,B 0,C 180,E1 -4446.559,E2 -4446.559} C_VEL
LIN {X 0,Y 530.991,Z 119.968,A -85,B 0,C 180,E1 -4449.444,E2 -4449.444} C_VEL
LIN {X 0,Y 530.967,Z 119.967,A -85,B 0,C 180,E1 -4452.458,E2 -4452.458} C_VEL
LIN {X 0,Y 530.979,Z 119.974,A -85,B 0,C 180,E1 -4455.623,E2 -4455.623} C_VEL
LIN {X 0,Y 530.996,Z 119.963,A -85,B 0,C 180,E1 -4458.565,E2 -4458.565} C_VEL
LIN {X 0,Y 530.958,Z 119.974,A -85,B 0,C 180,E1 -4461.53,E2 -4461.53} C_VEL
LIN {X 0,Y 530.957,Z 119.966,A -85,B 0,C 180,E1 -4464.38,E2 -4464.38} C_VEL
LIN {X 0,Y 530.969,Z 119.973,A -85,B 0,C 180,E1 -4467.134,E2 -4467.134} C_VEL
LIN {X 0,Y 530.954,Z 119.967,A -85,B 0,C 180,E1 -4469.802,E2 -4469.802} C_VEL
LIN {X 0,Y 530.974,Z 119.96,A -85,B 0,C 180,E1 -4472.477,E2 -4472.477} C_VEL
LIN {X 0,Y 530.959,Z 119.972,A -85,B 0,C 180,E1 -4474.94,E2 -4474.94} C_VEL
LIN {X 0,Y 530.98,Z 119.962,A -85,B 0,C 180,E1 -4477.899,E2 -4477.899} C_VEL
LIN {X 0,Y 530.985,Z 119.97,A -85,B 0,C 180,E1 -4480.677,E2 -4480.677} C_VEL
LIN {X 0,Y 530.962,Z 119.969,A -85,B 0,C 180,E1 -4483.07,E2 -4483.07} C_VEL
LIN {X 0,Y 531.004,Z 119.962,A -85,B 0,C 180,E1 -4485.436,E2 -4485.436} C_VEL
LIN {X 0,Y 531.039,Z 119.964,A -85,B 0,C 180,E1 -4488.55,E2 -4488.55} C_VEL
LIN {X 0,Y 531.034,Z 119.957,A -85,B 0,C 180,E1 -4491.629,E2 -4491.629} C_VEL
LIN {X 0,Y 531.088,Z 119.955,A -85,B 0,C 180,E1 -4494.685,E2 -4494.685} C_VEL
LIN {X 0,Y 531.137,Z 119.944,A -85,B 0,C 180,E1 -4497.725,E2 -4497.725} C_VEL
LIN {X 0,Y 531.132,Z 119.942,A -85,B 0,C 180,E1 -4500,E2 -4500} C_VEL
LIN {X 0,Y 531.137,Z 119.95,A -85,B 0,C 180,E1 -4502.275,E2 -4502.275} C_VEL
LIN {X 0,Y 531.085,Z 119.951,A -85,B 0,C 180,E1 -4505.315,E2 -4505.315} C_VEL
LIN {X 0,Y 530.986,Z 119.958,A -85,B 0,C 180,E1 -4508.372,E2 -4508.372} C_VEL
LIN {X 0,Y 531.016,Z 119.96,A -85,B 0,C 180,E1 -4511.65,E2 -4511.65} C_VEL
LIN {X 0,Y 530.968,Z 119.966,A -85,B 0,C 180,E1 -4514.928,E2 -4514.928} C_VEL
LIN {X 0,Y 530.949,Z 119.975,A -85,B 0,C 180,E1 -4517.725,E2 -4517.725} C_VEL
LIN {X 0,Y 530.93,Z 119.971,A -85,B 0,C 180,E1 -4520.941,E2 -4520.941} C_VEL
LIN {X 0,Y 530.924,Z 119.977,A -85,B 0,C 180,E1 -4523.399,E2 -4523.399} C_VEL
LIN {X 0,Y 530.926,Z 119.972,A -85,B 0,C 180,E1 -4525.902,E2 -4525.902} C_VEL
LIN {X 0,Y 530.934,Z 119.964,A -85,B 0,C 180,E1 -4528.46,E2 -4528.46} C_VEL
LIN {X 0,Y 530.94,Z 119.969,A -85,B 0,C 180,E1 -4531.081,E2 -4531.081} C_VEL
LIN {X 0,Y 530.937,Z 119.971,A -85,B 0,C 180,E1 -4533.777,E2 -4533.777} C_VEL
LIN {X 0,Y 530.909,Z 119.973,A -85,B 0,C 180,E1 -4536.563,E2 -4536.563} C_VEL
LIN {X 0,Y 530.958,Z 119.967,A -85,B 0,C 180,E1 -4539.447,E2 -4539.447} C_VEL
LIN {X 0,Y 530.92,Z 119.975,A -85,B 0,C 180,E1 -4542.463,E2 -4542.463} C_VEL
LIN {X 0,Y 530.93,Z 119.97,A -85,B 0,C 180,E1 -4543.522,E2 -4543.522} C_VEL
LIN {X 0,Y 530.265,Z 120.054,A -85,B 0,C 180,E1 -4544.156,E2 -4544.156} C_VEL
LIN {X 0,Y 527.427,Z 120.412,A -85,B 0,C 180,E1 -4545.185,E2 -4545.185} C_VEL
LIN {X 0,Y 525.021,Z 120.715,A -85,B 0,C 180,E1 -4546.013,E2 -4546.013} C_VEL
LIN {X 0,Y 523.975,Z 120.843,A -85,B 0,C 180,E1 -4546.653,E2 -4546.653} C_VEL
LIN {X 0,Y 523.883,Z 120.852,A -85,B 0,C 180,E1 -4546.869,E2 -4546.869} C_VEL
LIN {X 0,Y 523.918,Z 120.845,A -85,B 0,C 180,E1 -4549.917,E2 -4549.917} C_VEL
LIN {X 0,Y 523.909,Z 120.848,A -85,B 0,C 180,E1 -4552.867,E2 -4552.867} C_VEL
LIN {X 0,Y 523.917,Z 120.845,A -85,B 0,C 180,E1 -4555.708,E2 -4555.708} C_VEL
LIN {X 0,Y 523.923,Z 120.851,A -85,B 0,C 180,E1 -4558.455,E2 -4558.455} C_VEL
LIN {X 0,Y 523.91,Z 120.844,A -85,B 0,C 180,E1 -4561.123,E2 -4561.123} C_VEL
LIN {X 0,Y 523.917,Z 120.851,A -85,B 0,C 180,E1 -4563.997,E2 -4563.997} C_VEL
LIN {X 0,Y 523.913,Z 120.852,A -85,B 0,C 180,E1 -4566.269,E2 -4566.269} C_VEL
LIN {X 0,Y 523.95,Z 120.841,A -85,B 0,C 180,E1 -4568.766,E2 -4568.766} C_VEL
LIN {X 0,Y 523.941,Z 120.841,A -85,B 0,C 180,E1 -4571.22,E2 -4571.22} C_VEL
LIN {X 0,Y 523.917,Z 120.847,A -85,B 0,C 180,E1 -4573.638,E2 -4573.638} C_VEL
LIN {X 0,Y 523.932,Z 120.845,A -85,B 0,C 180,E1 -4576.027,E2 -4576.027} C_VEL
LIN {X 0,Y 524.019,Z 120.835,A -85,B 0,C 180,E1 -4578.394,E2 -4578.394} C_VEL
LIN {X 0,Y 523.991,Z 120.843,A -85,B 0,C 180,E1 -4581.515,E2 -4581.515} C_VEL
LIN {X 0,Y 524.061,Z 120.962,A -85,B 0,C 180,E1 -4584.203,E2 -4584.203} C_VEL
LIN {X 0,Y 526.032,Z 130.485,A -85,B 0,C 180,E1 -4585.786,E2 -4585.786} C_VEL
LIN {X 0,Y 525.777,Z 142.37,A -85,B 0,C 180,E1 -4587.57,E2 -4587.57} C_VEL
LIN {X 0,Y 528.56,Z 154.589,A -85,B 0,C 180,E1 -4587.865,E2 -4587.865} C_VEL
LIN {X 0,Y 527.592,Z 307.198,A -85,B 0,C 180,E1 -4590.024,E2 -4590.024} C_VEL
LIN {X 0,Y 527.313,Z 323.28,A -85,B 0,C 180,E1 -4590.419,E2 -4590.419} C_VEL
LIN {X 0,Y 526.926,Z 338.356,A -85,B 0,C 180,E1 -4590.955,E2 -4590.955} C_VEL
LIN {X 0,Y 526.514,Z 352.594,A -85,B 0,C 180,E1 -4591.625,E2 -4591.625} C_VEL
LIN {X 0,Y 526.051,Z 365.625,A -85,B 0,C 180,E1 -4592.392,E2 -4592.392} C_VEL
LIN {X 0,Y 525.543,Z 378.959,A -85,B 0,C 180,E1 -4593.354,E2 -4593.354} C_VEL
LIN {X 0,Y 525.029,Z 391.105,A -85,B 0,C 180,E1 -4594.414,E2 -4594.414} C_VEL
LIN {X 0,Y 524.679,Z 402.173,A -85,B 0,C 180,E1 -4595.573,E2 -4595.573} C_VEL
LIN {X 0,Y 524.332,Z 411.574,A -85,B 0,C 180,E1 -4596.735,E2 -4596.735} C_VEL
LIN {X 0,Y 523.996,Z 420.868,A -85,B 0,C 180,E1 -4598.096,E2 -4598.096} C_VEL
LIN {X 0,Y 523.757,Z 428.64,A -85,B 0,C 180,E1 -4599.461,E2 -4599.461} C_VEL
LIN {X 0,Y 523.56,Z 435.132,A -85,B 0,C 180,E1 -4600.832,E2 -4600.832} C_VEL
LIN {X 0,Y 523.447,Z 441.111,A -85,B 0,C 180,E1 -4602.405,E2 -4602.405} C_VEL
LIN {X 0,Y 523.381,Z 445.71,A -85,B 0,C 180,E1 -4603.987,E2 -4603.987} C_VEL
LIN {X 0,Y 523.261,Z 449.018,A -85,B 0,C 180,E1 -4605.582,E2 -4605.582} C_VEL
LIN {X 0,Y 523.291,Z 451.045,A -85,B 0,C 180,E1 -4607.185,E2 -4607.185} C_VEL
LIN {X 0,Y 523.266,Z 451.845,A -85,B 0,C 180,E1 -4608.805,E2 -4608.805} C_VEL
LIN {X 0,Y 523.257,Z 451.393,A -85,B 0,C 180,E1 -4610.439,E2 -4610.439} C_VEL
LIN {X 0,Y 523.303,Z 449.645,A -85,B 0,C 180,E1 -4612.089,E2 -4612.089} C_VEL
LIN {X 0,Y 523.345,Z 446.516,A -85,B 0,C 180,E1 -4613.757,E2 -4613.757} C_VEL
LIN {X 0,Y 523.451,Z 441.886,A -85,B 0,C 180,E1 -4615.445,E2 -4615.445} C_VEL
LIN {X 0,Y 523.536,Z 437.353,A -85,B 0,C 180,E1 -4616.725,E2 -4616.725} C_VEL
LIN {X 0,Y 523.729,Z 430.72,A -85,B 0,C 180,E1 -4618.231,E2 -4618.231} C_VEL
LIN {X 0,Y 523.957,Z 422.405,A -85,B 0,C 180,E1 -4619.755,E2 -4619.755} C_VEL
LIN {X 0,Y 524.254,Z 413.017,A -85,B 0,C 180,E1 -4621.17,E2 -4621.17} C_VEL
LIN {X 0,Y 524.663,Z 402.871,A -85,B 0,C 180,E1 -4622.445,E2 -4622.445} C_VEL
LIN {X 0,Y 525.094,Z 391.009,A -85,B 0,C 180,E1 -4623.687,E2 -4623.687} C_VEL
LIN {X 0,Y 525.569,Z 378.824,A -85,B 0,C 180,E1 -4624.749,E2 -4624.749} C_VEL
LIN {X 0,Y 526.061,Z 365.193,A -85,B 0,C 180,E1 -4625.728,E2 -4625.728} C_VEL
LIN {X 0,Y 526.538,Z 352.039,A -85,B 0,C 180,E1 -4626.498,E2 -4626.498} C_VEL
LIN {X 0,Y 526.94,Z 337.299,A -85,B 0,C 180,E1 -4627.182,E2 -4627.182} C_VEL
LIN {X 0,Y 527.314,Z 321.627,A -85,B 0,C 180,E1 -4627.722,E2 -4627.722} C_VEL
LIN {X 0,Y 527.594,Z 306.639,A -85,B 0,C 180,E1 -4628.077,E2 -4628.077} C_VEL
LIN {X 0,Y 528.528,Z 154.549,A -85,B 0,C 180,E1 -4630.228,E2 -4630.228} C_VEL
LIN {X 0,Y 525.751,Z 142.152,A -85,B 0,C 180,E1 -4630.547,E2 -4630.547} C_VEL
LIN {X 0,Y 526.02,Z 130.665,A -85,B 0,C 180,E1 -4632.309,E2 -4632.309} C_VEL
LIN {X 0,Y 523.943,Z 120.847,A -85,B 0,C 180,E1 -4633.97,E2 -4633.97} C_VEL
LIN {X 0,Y 523.903,Z 120.854,A -85,B 0,C 180,E1 -4636.831,E2 -4636.831} C_VEL
LIN {X 0,Y 523.94,Z 120.848,A -85,B 0,C 180,E1 -4639.87,E2 -4639.87} C_VEL
LIN {X 0,Y 523.906,Z 120.85,A -85,B 0,C 180,E1 -4642.867,E2 -4642.867} C_VEL
LIN {X 0,Y 523.933,Z 120.842,A -85,B 0,C 180,E1 -4645.709,E2 -4645.709} C_VEL
LIN {X 0,Y 523.921,Z 120.848,A -85,B 0,C 180,E1 -4648.455,E2 -4648.455} C_VEL
LIN {X 0,Y 523.929,Z 120.841,A -85,B 0,C 180,E1 -4651.124,E2 -4651.124} C_VEL
LIN {X 0,Y 523.925,Z 120.852,A -85,B 0,C 180,E1 -4653.993,E2 -4653.993} C_VEL
LIN {X 0,Y 523.91,Z 120.847,A -85,B 0,C 180,E1 -4656.269,E2 -4656.269} C_VEL
LIN {X 0,Y 523.947,Z 120.841,A -85,B 0,C 180,E1 -4658.766,E2 -4658.766} C_VEL
LIN {X 0,Y 523.938,Z 120.843,A -85,B 0,C 180,E1 -4661.22,E2 -4661.22} C_VEL
LIN {X 0,Y 523.919,Z 120.85,A -85,B 0,C 180,E1 -4663.638,E2 -4663.638} C_VEL
LIN {X 0,Y 523.929,Z 120.848,A -85,B 0,C 180,E1 -4666.027,E2 -4666.027} C_VEL
LIN {X 0,Y 524.014,Z 120.832,A -85,B 0,C 180,E1 -4668.394,E2 -4668.394} C_VEL
LIN {X 0,Y 524,Z 120.839,A -85,B 0,C 180,E1 -4671.516,E2 -4671.516} C_VEL
LIN {X 0,Y 524.08,Z 120.822,A -85,B 0,C 180,E1 -4674.613,E2 -4674.613} C_VEL
LIN {X 0,Y 524.114,Z 120.823,A -85,B 0,C 180,E1 -4677.694,E2 -4677.694} C_VEL
LIN {X 0,Y 524.12,Z 120.82,A -85,B 0,C 180,E1 -4680.768,E2 -4680.768} C_VEL
LIN {X 0,Y 524.068,Z 120.83,A -85,B 0,C 180,E1 -4683.075,E2 -4683.075} C_VEL
LIN {X 0,Y 524.034,Z 120.829,A -85,B 0,C 180,E1 -4686.159,E2 -4686.159} C_VEL
LIN {X 0,Y 523.987,Z 120.841,A -85,B 0,C 180,E1 -4689.262,E2 -4689.262} C_VEL
LIN {X 0,Y 524.003,Z 120.833,A -85,B 0,C 180,E1 -4691.739,E2 -4691.739} C_VEL
LIN {X 0,Y 523.993,Z 120.841,A -85,B 0,C 180,E1 -4695.052,E2 -4695.052} C_VEL
LIN {X 0,Y 523.947,Z 120.841,A -85,B 0,C 180,E1 -4697.969,E2 -4697.969} C_VEL
LIN {X 0,Y 523.971,Z 120.838,A -85,B 0,C 180,E1 -4700.41,E2 -4700.41} C_VEL
LIN {X 0,Y 523.91,Z 120.851,A -85,B 0,C 180,E1 -4702.893,E2 -4702.893} C_VEL
LIN {X 0,Y 523.952,Z 120.84,A -85,B 0,C 180,E1 -4705.418,E2 -4705.418} C_VEL
LIN {X 0,Y 523.964,Z 120.84,A -85,B 0,C 180,E1 -4707.999,E2 -4707.999} C_VEL
LIN {X 0,Y 523.943,Z 120.846,A -85,B 0,C 180,E1 -4710.855,E2 -4710.855} C_VEL
LIN {X 0,Y 523.929,Z 120.844,A -85,B 0,C 180,E1 -4713.73,E2 -4713.73} C_VEL
LIN {X 0,Y 523.903,Z 120.854,A -85,B 0,C 180,E1 -4716.401,E2 -4716.401} C_VEL
LIN {X 0,Y 523.919,Z 120.842,A -85,B 0,C 180,E1 -4719.085,E2 -4719.085} C_VEL
LIN {X 0,Y 523.95,Z 120.847,A -85,B 0,C 180,E1 -4722.119,E2 -4722.119} C_VEL
LIN {X 0,Y 523.955,Z 120.84,A -85,B 0,C 180,E1 -4725.309,E2 -4725.309} C_VEL
LIN {X 0,Y 523.954,Z 120.842,A -85,B 0,C 180,E1 -4728.69,E2 -4728.69} C_VEL
LIN {X 0,Y 523.919,Z 120.846,A -85,B 0,C 180,E1 -4731.08,E2 -4731.08} C_VEL
LIN {X 0,Y 523.899,Z 120.853,A -85,B 0,C 180,E1 -4733.825,E2 -4733.825} C_VEL
LIN {X 0,Y 523.94,Z 120.842,A -85,B 0,C 180,E1 -4736.636,E2 -4736.636} C_VEL
LIN {X 0,Y 523.955,Z 120.844,A -85,B 0,C 180,E1 -4739.356,E2 -4739.356} C_VEL
LIN {X 0,Y 523.991,Z 120.921,A -85,B 0,C 180,E1 -4742.003,E2 -4742.003} C_VEL
LIN {X 0,Y 526.761,Z 133.496,A -85,B 0,C 180,E1 -4743.878,E2 -4743.878} C_VEL
LIN {X 0,Y 526.121,Z 155.477,A -85,B 0,C 180,E1 -4746.793,E2 -4746.793} C_VEL
LIN {X 0,Y 525.728,Z 168.893,A -85,B 0,C 180,E1 -4748.51,E2 -4748.51} C_VEL
LIN {X 0,Y 528.51,Z 183.996,A -85,B 0,C 180,E1 -4748.843,E2 -4748.843} C_VEL
LIN {X 0,Y 527.534,Z 334.549,A -85,B 0,C 180,E1 -4750.966,E2 -4750.966} C_VEL
LIN {X 0,Y 527.225,Z 349.524,A -85,B 0,C 180,E1 -4751.319,E2 -4751.319} C_VEL
LIN {X 0,Y 526.889,Z 364.552,A -85,B 0,C 180,E1 -4751.833,E2 -4751.833} C_VEL
LIN {X 0,Y 526.419,Z 377.654,A -85,B 0,C 180,E1 -4752.419,E2 -4752.419} C_VEL
LIN {X 0,Y 525.957,Z 391.629,A -85,B 0,C 180,E1 -4753.205,E2 -4753.205} C_VEL
LIN {X 0,Y 525.488,Z 404.944,A -85,B 0,C 180,E1 -4754.127,E2 -4754.127} C_VEL
LIN {X 0,Y 524.991,Z 417.387,A -85,B 0,C 180,E1 -4755.169,E2 -4755.169} C_VEL
LIN {X 0,Y 524.607,Z 428.188,A -85,B 0,C 180,E1 -4756.244,E2 -4756.244} C_VEL
LIN {X 0,Y 524.268,Z 438.207,A -85,B 0,C 180,E1 -4757.418,E2 -4757.418} C_VEL
LIN {X 0,Y 523.941,Z 448.005,A -85,B 0,C 180,E1 -4758.785,E2 -4758.785} C_VEL
LIN {X 0,Y 523.706,Z 456.182,A -85,B 0,C 180,E1 -4760.148,E2 -4760.148} C_VEL
LIN {X 0,Y 523.58,Z 462.938,A -85,B 0,C 180,E1 -4761.509,E2 -4761.509} C_VEL
LIN {X 0,Y 523.48,Z 469.18,A -85,B 0,C 180,E1 -4763.06,E2 -4763.06} C_VEL
LIN {X 0,Y 523.442,Z 474.007,A -85,B 0,C 180,E1 -4764.607,E2 -4764.607} C_VEL
LIN {X 0,Y 523.384,Z 477.542,A -85,B 0,C 180,E1 -4766.151,E2 -4766.151} C_VEL
LIN {X 0,Y 523.332,Z 479.867,A -85,B 0,C 180,E1 -4767.691,E2 -4767.691} C_VEL
LIN {X 0,Y 523.246,Z 481.036,A -85,B 0,C 180,E1 -4769.231,E2 -4769.231} C_VEL
LIN {X 0,Y 523.246,Z 481.036,A -85,B 0,C 180,E1 -4770.77,E2 -4770.77} C_VEL
LIN {X 0,Y 523.332,Z 479.866,A -85,B 0,C 180,E1 -4772.309,E2 -4772.309} C_VEL
LIN {X 0,Y 523.384,Z 477.543,A -85,B 0,C 180,E1 -4773.85,E2 -4773.85} C_VEL
LIN {X 0,Y 523.442,Z 474.016,A -85,B 0,C 180,E1 -4775.393,E2 -4775.393} C_VEL
LIN {X 0,Y 523.49,Z 469.195,A -85,B 0,C 180,E1 -4776.94,E2 -4776.94} C_VEL
LIN {X 0,Y 523.581,Z 462.95,A -85,B 0,C 180,E1 -4778.491,E2 -4778.491} C_VEL
LIN {X 0,Y 523.773,Z 455.107,A -85,B 0,C 180,E1 -4780.046,E2 -4780.046} C_VEL
LIN {X 0,Y 524.005,Z 446.765,A -85,B 0,C 180,E1 -4781.41,E2 -4781.41} C_VEL
LIN {X 0,Y 524.313,Z 436.713,A -85,B 0,C 180,E1 -4782.778,E2 -4782.778} C_VEL
LIN {X 0,Y 524.687,Z 426.436,A -85,B 0,C 180,E1 -4783.952,E2 -4783.952} C_VEL
LIN {X 0,Y 525.156,Z 414.335,A -85,B 0,C 180,E1 -4785.114,E2 -4785.114} C_VEL
LIN {X 0,Y 525.597,Z 401.896,A -85,B 0,C 180,E1 -4786.109,E2 -4786.109} C_VEL
LIN {X 0,Y 526.106,Z 388.512,A -85,B 0,C 180,E1 -4786.991,E2 -4786.991} C_VEL
LIN {X 0,Y 526.508,Z 375.73,A -85,B 0,C 180,E1 -4787.679,E2 -4787.679} C_VEL
LIN {X 0,Y 526.964,Z 362.04,A -85,B 0,C 180,E1 -4788.266,E2 -4788.266} C_VEL
LIN {X 0,Y 527.303,Z 347.296,A -85,B 0,C 180,E1 -4788.743,E2 -4788.743} C_VEL
LIN {X 0,Y 527.524,Z 333.117,A -85,B 0,C 180,E1 -4789.061,E2 -4789.061} C_VEL
LIN {X 0,Y 528.522,Z 183.584,A -85,B 0,C 180,E1 -4791.164,E2 -4791.164} C_VEL
LIN {X 0,Y 525.706,Z 168.549,A -85,B 0,C 180,E1 -4791.521,E2 -4791.521} C_VEL
LIN {X 0,Y 526.322,Z 149.327,A -85,B 0,C 180,E1 -4794.034,E2 -4794.034} C_VEL
LIN {X 0,Y 526.81,Z 133.594,A -85,B 0,C 180,E1 -4796.12,E2 -4796.12} C_VEL
LIN {X 0,Y 523.973,Z 120.845,A -85,B 0,C 180,E1 -4798.026,E2 -4798.026} C_VEL
LIN {X 0,Y 523.946,Z 120.843,A -85,B 0,C 180,E1 -4800.855,E2 -4800.855} C_VEL
LIN {X 0,Y 523.961,Z 120.848,A -85,B 0,C 180,E1 -4803.735,E2 -4803.735} C_VEL
LIN {X 0,Y 523.905,Z 120.85,A -85,B 0,C 180,E1 -4806.402,E2 -4806.402} C_VEL
LIN {X 0,Y 523.924,Z 120.845,A -85,B 0,C 180,E1 -4809.085,E2 -4809.085} C_VEL
LIN {X 0,Y 523.945,Z 120.844,A -85,B 0,C 180,E1 -4812.12,E2 -4812.12} C_VEL
LIN {X 0,Y 523.946,Z 120.847,A -85,B 0,C 180,E1 -4815.311,E2 -4815.311} C_VEL
LIN {X 0,Y 523.958,Z 120.841,A -85,B 0,C 180,E1 -4818.69,E2 -4818.69} C_VEL
